END_VAR
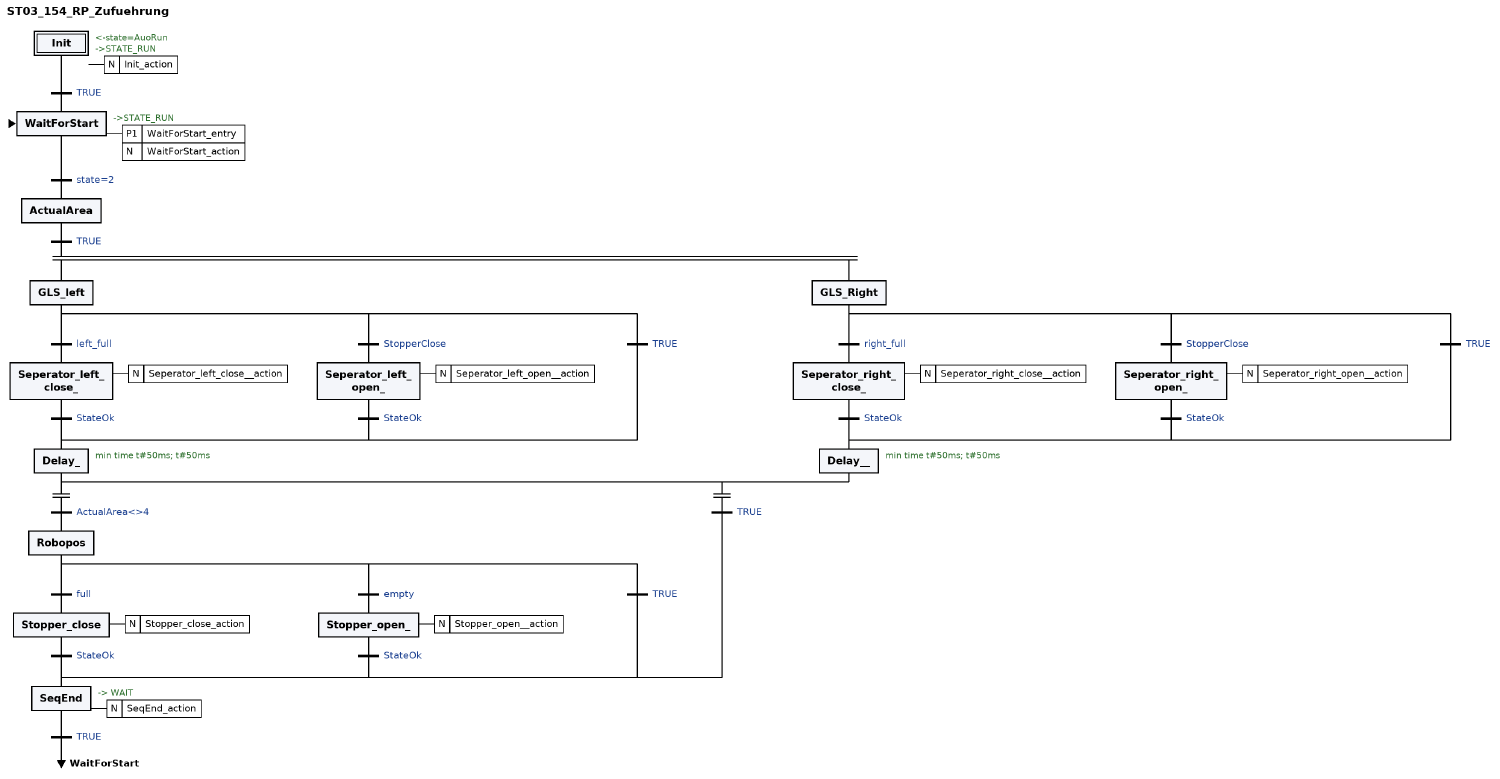
[picture p57: ST03_154_RP_Zufuehrung (SFC)]
INITIAL_STEP Init: (* <-state=AuoRun / ->STATE_RUN *)
	Init_action(N);
END_STEP
TRANSITION FROM Init TO WaitForStart := TRUE;
END_TRANSITION
STEP WaitForStart: (* ->STATE_RUN *)
	WaitForStart_entry(P1);
	WaitForStart_action(N);
END_STEP
TRANSITION FROM WaitForStart TO ActualArea := state=2;
END_TRANSITION
STEP ActualArea:
END_STEP
TRANSITION FROM ActualArea TO (GLS_left, GLS_Right) := TRUE;
END_TRANSITION
STEP GLS_left:
END_STEP
TRANSITION FROM GLS_left TO Seperator_left_close_ := left_full;
END_TRANSITION
TRANSITION FROM GLS_left TO Seperator_left_open_ := StopperClose;
END_TRANSITION
TRANSITION FROM GLS_left TO Delay_ := TRUE;
END_TRANSITION
STEP Seperator_left_close_:
	Seperator_left_close__action(N);
END_STEP
TRANSITION FROM Seperator_left_close_ TO Delay_ := StateOk;
END_TRANSITION
STEP Seperator_left_open_:
	Seperator_left_open__action(N);
END_STEP
TRANSITION FROM Seperator_left_open_ TO Delay_ := StateOk;
END_TRANSITION
STEP Delay_: (* min time t#50ms; t#50ms *)
END_STEP
STEP GLS_Right:
END_STEP
TRANSITION FROM GLS_Right TO Seperator_right_close_ := right_full;
END_TRANSITION
TRANSITION FROM GLS_Right TO Seperator_right_open_ := StopperClose;
END_TRANSITION
TRANSITION FROM GLS_Right TO Delay__ := TRUE;
END_TRANSITION
STEP Seperator_right_close_:
	Seperator_right_close__action(N);
END_STEP
TRANSITION FROM Seperator_right_close_ TO Delay__ := StateOk;
END_TRANSITION
STEP Seperator_right_open_:
	Seperator_right_open__action(N);
END_STEP
TRANSITION FROM Seperator_right_open_ TO Delay__ := StateOk;
END_TRANSITION
STEP Delay__: (* min time t#50ms; t#50ms *)
END_STEP
TRANSITION FROM (Delay_, Delay__) TO Robopos := ActualArea<>4;
END_TRANSITION
TRANSITION FROM (Delay_, Delay__) TO SeqEnd := TRUE;
END_TRANSITION
STEP Robopos:
END_STEP
TRANSITION FROM Robopos TO Stopper_close := full;
END_TRANSITION
TRANSITION FROM Robopos TO Stopper_open_ := empty;
END_TRANSITION
TRANSITION FROM Robopos TO SeqEnd := TRUE;
END_TRANSITION
STEP Stopper_close:
	Stopper_close_action(N);
END_STEP
TRANSITION FROM Stopper_close TO SeqEnd := StateOk;
END_TRANSITION
STEP Stopper_open_:
	Stopper_open__action(N);
END_STEP
TRANSITION FROM Stopper_open_ TO SeqEnd := StateOk;
END_TRANSITION
STEP SeqEnd: (* -> WAIT *)
	SeqEnd_action(N);
END_STEP
TRANSITION FROM SeqEnd TO WaitForStart := TRUE;
END_TRANSITION

ACTION Init_action:
Start:=FALSE;
State:=STATE_WAIT;
MsgOK:=FALSE;
MsgCancel:=FALSE;
SFCRun:=FALSE;
Result:=RESULT_NON;
END_ACTION

ACTION WaitForStart_entry:
;
END_ACTION

ACTION WaitForStart_action:
IF 	Start   THEN
	State:=STATE_RUN;
	Result:=RESULT_NON;
	SFCTimeStart:=TIME();
	Start:=FALSE;
ELSE
	State:=STATE_WAIT;
	MsgOK:=FALSE;
	MsgCancel:=FALSE;
	SFCRun:=FALSE;
END_IF
END_ACTION

ACTION Seperator_left_close__action:
ST03_419_Y61_5.MoveWork:=TRUE;	(* Förderband linke Zuführung Vereinzler AST/GST *)
END_ACTION

ACTION Seperator_left_open__action:
ST03_419_Y61_5.MoveInit:=TRUE;		(* Förderband linke Zuführung Vereinzler AST/GST *)
END_ACTION

ACTION Seperator_right_close__action:
ST03_419_Y61_6.MoveWork:=TRUE;	(* Förderband rechts Zuführung Vereinzler AST/GST *)
END_ACTION

ACTION Seperator_right_open__action:
ST03_419_Y61_6.MoveInit:=TRUE;			(* Förderband rechts Zuführung Vereinzler AST/GST *)
END_ACTION

ACTION Stopper_close_action:
ST03_419_Y61_7.MoveInit:=TRUE;		(* Förderband links/rechts Züführung Stopper AST/GST *)
END_ACTION

ACTION Stopper_open__action:
ST03_419_Y61_7.MoveWork:=TRUE;		(* Förderband links/rechts Züführung Stopper AST/GST *)
END_ACTION

ACTION SeqEnd_action:
SFCTime:=TIME_TO_DINT(TIME()-SFCTimeStart);
State:=STATE_WAIT;
END_ACTION

TRANSITION left_full:
ST03_419_B61_0.BitInToCheck			(*  Förderband Zuführung links ISK anwesend zum Vereinzeln*)
END_TRANSITION

TRANSITION StateOk:
ST03_419_Y61_5.State=STATE_OK
AND
gTipImp
END_TRANSITION

TRANSITION StopperClose:
NOT ST03_418_B60_4.ValveSensor AND
ST03_418_B60_5.ValveSensor
END_TRANSITION

TRANSITION StateOk:
ST03_419_Y61_5.State=STATE_OK 	(* Förderband  Zuführung Vereinzler AST/GST *)
AND
gTipImp
END_TRANSITION

TRANSITION right_full:
ST03_419_B61_1.BitInToCheck			(*  Förderband Zuführung rechts ISK anwesend zum Vereinzeln*)
END_TRANSITION

TRANSITION StateOk:
ST03_419_Y61_6.State=STATE_OK (* Förderband rechts Zuführung Vereinzler AST/GST *)
AND
gTipImp
END_TRANSITION

TRANSITION StopperClose:
NOT ST03_418_B60_4.ValveSensor AND
ST03_418_B60_5.ValveSensor
END_TRANSITION

TRANSITION StateOk:
ST03_419_Y61_6.State=STATE_OK 	(* Förderband rechts Zuführung Vereinzler AST/GST *)
AND
gTipImp
END_TRANSITION

TRANSITION ActualArea<>4:
Robot01.ActualArea <> 4
END_TRANSITION

TRANSITION full:
ST03_419_B61_2.BitInToCheck AND 	(*  Züführung links ISK auf Übergabeposition Roboter Palettierer*)
ST03_419_B61_3.BitInToCheck		(*  Züführung rechts ISK auf Übergabeposition Roboter Palettierer*)
END_TRANSITION

TRANSITION StateOk:
ST03_419_Y61_7.State=STATE_OK 	(* Förderband  Zuführung Vereinzler AST/GST *)
AND
gTipImp
END_TRANSITION

TRANSITION empty:
NOT ST03_419_B61_2.BitInToCheck AND 	(*  Züführung links ISK auf Übergabeposition Roboter Palettierer*)
NOT ST03_419_B61_3.BitInToCheck		(*  Züführung rechts ISK auf Übergabeposition Roboter Palettierer*)
END_TRANSITION

TRANSITION StateOk:
ST03_419_Y61_7.State=STATE_OK 	(* Förderband  Zuführung Vereinzler AST/GST *)
AND
gTipImp
END_TRANSITION
END_PROGRAM

(* POU Stations/ST_03_Ruestsaetze/ST_03_SFCs/Zufuehrungen/ST03_206pol_Zufuehrung, SFC *)
 PROGRAM ST03_206pol_Zufuehrung
VAR_OUTPUT
	SFCCurrentPOU			: STRING:='ST03_206pol_Zufuehrung';
	SFCCurrentStep			: STRING:='';
	FB_CurrentStepHistorie	: FB_CurrentStepHistorie;
	SFCTime					: DINT;
	State   				: StateObject	:= STATE_WAIT;
	Result  				: StateResult;
END_VAR
VAR_INPUT
	Start					:BOOL;
END_VAR
VAR
	MsgOK				: BOOL;
	MsgCancel			: BOOL;
	SFCRun				: BOOL;
	SFCTimeStart		: TIME;
	Delay				: TON;
	(* Userdefinded area *)

END_VAR
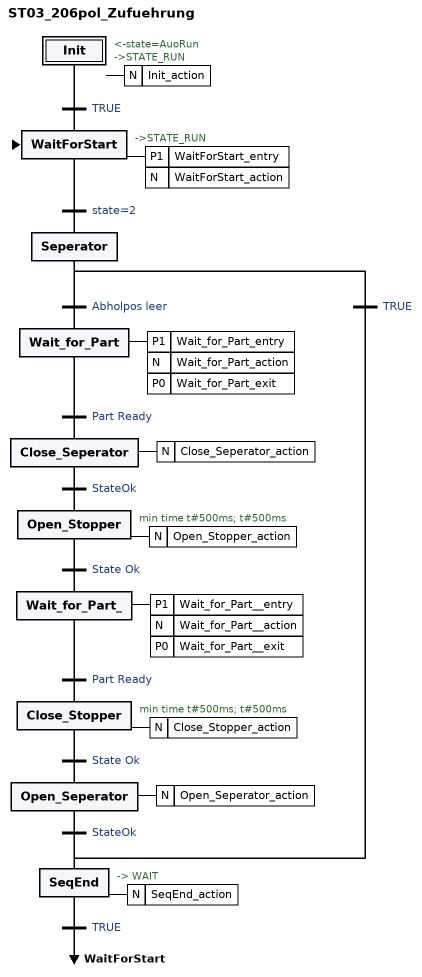
INITIAL_STEP Init: (* <-state=AuoRun / ->STATE_RUN *)
	Init_action(N);
END_STEP
TRANSITION FROM Init TO WaitForStart := TRUE;
END_TRANSITION
STEP WaitForStart: (* ->STATE_RUN *)
	WaitForStart_entry(P1);
	WaitForStart_action(N);
END_STEP
TRANSITION FROM WaitForStart TO Seperator := state=2;
END_TRANSITION
STEP Seperator:
END_STEP
TRANSITION FROM Seperator TO Wait_for_Part := Abholpos leer;
END_TRANSITION
TRANSITION FROM Seperator TO SeqEnd := TRUE;
END_TRANSITION
STEP Wait_for_Part:
	Wait_for_Part_entry(P1);
	Wait_for_Part_action(N);
	Wait_for_Part_exit(P0);
END_STEP
TRANSITION FROM Wait_for_Part TO Close_Seperator := Part Ready;
END_TRANSITION
STEP Close_Seperator:
	Close_Seperator_action(N);
END_STEP
TRANSITION FROM Close_Seperator TO Open_Stopper := StateOk;
END_TRANSITION
STEP Open_Stopper: (* min time t#500ms; t#500ms *)
	Open_Stopper_action(N);
END_STEP
TRANSITION FROM Open_Stopper TO Wait_for_Part_ := State Ok;
END_TRANSITION
STEP Wait_for_Part_:
	Wait_for_Part__entry(P1);
	Wait_for_Part__action(N);
	Wait_for_Part__exit(P0);
END_STEP
TRANSITION FROM Wait_for_Part_ TO Close_Stopper := Part Ready;
END_TRANSITION
STEP Close_Stopper: (* min time t#500ms; t#500ms *)
	Close_Stopper_action(N);
END_STEP
TRANSITION FROM Close_Stopper TO Open_Seperator := State Ok;
END_TRANSITION
STEP Open_Seperator:
	Open_Seperator_action(N);
END_STEP
TRANSITION FROM Open_Seperator TO SeqEnd := StateOk;
END_TRANSITION
STEP SeqEnd: (* -> WAIT *)
	SeqEnd_action(N);
END_STEP
TRANSITION FROM SeqEnd TO WaitForStart := TRUE;
END_TRANSITION

ACTION Init_action:
Start:=FALSE;
State:=STATE_WAIT;
MsgOK:=FALSE;
MsgCancel:=FALSE;
SFCRun:=FALSE;
Result:=RESULT_NON;
END_ACTION

ACTION WaitForStart_entry:
;
END_ACTION

ACTION WaitForStart_action:
IF 	Start   THEN
	State:=STATE_RUN;
	Result:=RESULT_NON;
	SFCTimeStart:=TIME();
	Start:=FALSE;
ELSE
	State:=STATE_WAIT;
	MsgOK:=FALSE;
	MsgCancel:=FALSE;
	SFCRun:=FALSE;
END_IF
END_ACTION

ACTION Wait_for_Part_entry:
ProcessMessage01:='';
Delay.IN:=FALSE;
Delay();
END_ACTION

ACTION Wait_for_Part_action:
ProcessMessage01:='1IM6';(*warte auf Teil in Vereinzelung*)
Delay.IN:=ST03_435_B67_7.BitInToCheck; 		 (* Schnittstelle Iso auf Übergabeposition *)
Delay.PT:=T#500ms;
Delay();
END_ACTION

ACTION Wait_for_Part_exit:
ProcessMessage01:='';
END_ACTION

ACTION Close_Seperator_action:
ST03_437_Y68_5.MoveWork:=TRUE;		(* Förderband  Zuführung Vereinzler AST/GST *)
END_ACTION

ACTION Open_Stopper_action:
ST03_437_Y68_6.MoveWork:=TRUE;		(* Förderband  Züführung Stopper AST/GST *)
END_ACTION

ACTION Wait_for_Part__entry:
ProcessMessage01:='';
Delay.IN:=FALSE;
Delay();
END_ACTION

ACTION Wait_for_Part__action:
ProcessMessage01:='1IM6';(*warte auf Teil in Vereinzelung*)
Delay.IN:=	ST03_Init_AbholPos.RoboPos31 OR
			ST03_Init_AbholPos.RoboPos35 OR
			NOT ST03_437_B68_4.BitInToCheck;
Delay.PT:=T#500ms;
Delay();
END_ACTION

ACTION Wait_for_Part__exit:
ProcessMessage01:='';
END_ACTION

ACTION Close_Stopper_action:
ST03_437_Y68_6.MoveInit:=TRUE;		(* Förderband  Züführung Stopper AST/GST *)
END_ACTION

ACTION Open_Seperator_action:
ST03_437_Y68_5.MoveInit:=TRUE;		(* Förderband  Zuführung Vereinzler AST/GST *)
END_ACTION

ACTION SeqEnd_action:
SFCTime:=TIME_TO_DINT(TIME()-SFCTimeStart);
State:=STATE_WAIT;
END_ACTION

TRANSITION Abholpos leer:
NOT ST03_Init_AbholPos.RoboPos31 AND
NOT ST03_Init_AbholPos.RoboPos35
END_TRANSITION

TRANSITION Part Ready:
Delay.Q AND
ST03_435_B67_7.BitInToCheck	AND	(*  ISK anwesend am Stoper*)
Robot01.ActualArea <> 4
END_TRANSITION

TRANSITION StateOk:
ST03_437_Y68_5.State=STATE_OK 	(* Förderband  Zuführung Vereinzler AST/GST *)

(*ST03_426_B68_4.BitInToCheck	AND		(*  Züführung  ISK auf Übergabeposition Roboter Palettierer*)
NOT ST03_425_B67_7.BitInToCheck AND	(*  ISK anwesend am Vereinzler*)
gTipImp*)
END_TRANSITION

TRANSITION State Ok:
ST03_437_Y68_6.State=STATE_OK 	(* Förderband  Züführung Stopper AST/GST *)
END_TRANSITION

TRANSITION Part Ready:
Delay.Q AND
(ST03_Init_AbholPos.RoboPos31 OR
ST03_Init_AbholPos.RoboPos35) AND
Robot01.ActualArea <> 4
END_TRANSITION

TRANSITION State Ok:
ST03_437_Y68_6.State=STATE_OK 	(* Förderband  Züführung Stopper AST/GST *)
END_TRANSITION

TRANSITION StateOk:
ST03_437_Y68_5.State=STATE_OK 	(* Förderband  Zuführung Vereinzler AST/GST *)
END_TRANSITION
END_PROGRAM

(* POU Stations/ST_03_Ruestsaetze/ST_03_SFCs/Zufuehrungen/ST03_92pol_Zufuehrung, SFC *)
 PROGRAM ST03_92pol_Zufuehrung
VAR_OUTPUT
	SFCCurrentPOU			: STRING:='ST03_92pol_Zufuehrung';
	SFCCurrentStep			: STRING:='';
	FB_CurrentStepHistorie	: FB_CurrentStepHistorie;
	SFCTime					: DINT;
	State   				: StateObject	:= STATE_WAIT;
	Result  				: StateResult;
END_VAR
VAR_INPUT
	Start					:BOOL;
END_VAR
VAR
	MsgOK				: BOOL;
	MsgCancel			: BOOL;
	SFCRun				: BOOL;
	SFCTimeStart		: TIME;
	Delay				: TON;
	(* Userdefinded area *)

END_VAR
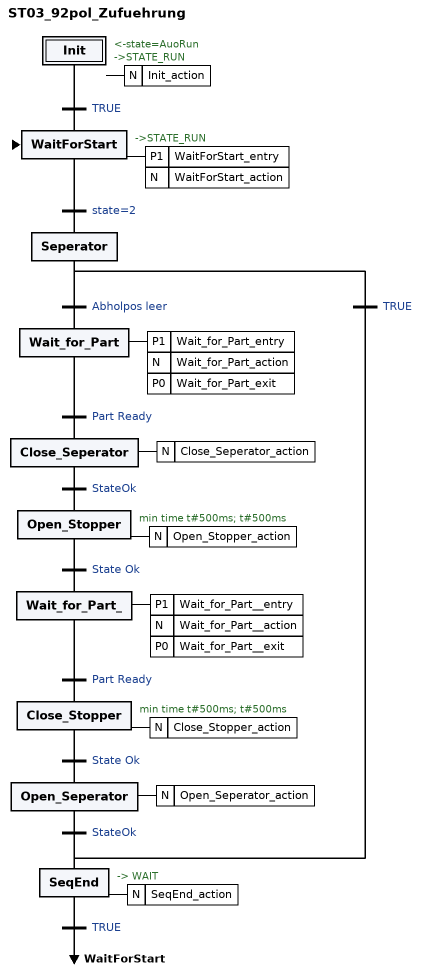
INITIAL_STEP Init: (* <-state=AuoRun / ->STATE_RUN *)
	Init_action(N);
END_STEP
TRANSITION FROM Init TO WaitForStart := TRUE;
END_TRANSITION
STEP WaitForStart: (* ->STATE_RUN *)
	WaitForStart_entry(P1);
	WaitForStart_action(N);
END_STEP
TRANSITION FROM WaitForStart TO Seperator := state=2;
END_TRANSITION
STEP Seperator:
END_STEP
TRANSITION FROM Seperator TO Wait_for_Part := Abholpos leer;
END_TRANSITION
TRANSITION FROM Seperator TO SeqEnd := TRUE;
END_TRANSITION
STEP Wait_for_Part:
	Wait_for_Part_entry(P1);
	Wait_for_Part_action(N);
	Wait_for_Part_exit(P0);
END_STEP
TRANSITION FROM Wait_for_Part TO Close_Seperator := Part Ready;
END_TRANSITION
STEP Close_Seperator:
	Close_Seperator_action(N);
END_STEP
TRANSITION FROM Close_Seperator TO Open_Stopper := StateOk;
END_TRANSITION
STEP Open_Stopper: (* min time t#500ms; t#500ms *)
	Open_Stopper_action(N);
END_STEP
TRANSITION FROM Open_Stopper TO Wait_for_Part_ := State Ok;
END_TRANSITION
STEP Wait_for_Part_:
	Wait_for_Part__entry(P1);
	Wait_for_Part__action(N);
	Wait_for_Part__exit(P0);
END_STEP
TRANSITION FROM Wait_for_Part_ TO Close_Stopper := Part Ready;
END_TRANSITION
STEP Close_Stopper: (* min time t#500ms; t#500ms *)
	Close_Stopper_action(N);
END_STEP
TRANSITION FROM Close_Stopper TO Open_Seperator := State Ok;
END_TRANSITION
STEP Open_Seperator:
	Open_Seperator_action(N);
END_STEP
TRANSITION FROM Open_Seperator TO SeqEnd := StateOk;
END_TRANSITION
STEP SeqEnd: (* -> WAIT *)
	SeqEnd_action(N);
END_STEP
TRANSITION FROM SeqEnd TO WaitForStart := TRUE;
END_TRANSITION

ACTION Init_action:
Start:=FALSE;
State:=STATE_WAIT;
MsgOK:=FALSE;
MsgCancel:=FALSE;
SFCRun:=FALSE;
Result:=RESULT_NON;
END_ACTION

ACTION WaitForStart_entry:
;
END_ACTION

ACTION WaitForStart_action:
IF 	Start   THEN
	State:=STATE_RUN;
	Result:=RESULT_NON;
	SFCTimeStart:=TIME();
	Start:=FALSE;
ELSE
	State:=STATE_WAIT;
	MsgOK:=FALSE;
	MsgCancel:=FALSE;
	SFCRun:=FALSE;
END_IF
END_ACTION

ACTION Wait_for_Part_entry:
ProcessMessage01:='';
Delay.IN:=FALSE;
Delay();
END_ACTION

ACTION Wait_for_Part_action:
ProcessMessage01:='1IM6';(*warte auf Teil in Vereinzelung*)
Delay.IN:=ST03_444_B69_7.BitInToCheck; 		 (* Schnittstelle Iso auf Übergabeposition *)
Delay.PT:=T#500ms;
Delay();
END_ACTION

ACTION Wait_for_Part_exit:
ProcessMessage01:='';
END_ACTION

ACTION Close_Seperator_action:
ST03_446_Y70_5.MoveWork:=TRUE;		(* Förderband  Zuführung Vereinzler AST/GST *)
END_ACTION

ACTION Open_Stopper_action:
ST03_446_Y70_6.MoveWork:=TRUE;		(* Förderband  Züführung Stopper AST/GST *)
END_ACTION

ACTION Wait_for_Part__entry:
ProcessMessage01:='';
Delay.IN:=FALSE;
Delay();
END_ACTION

ACTION Wait_for_Part__action:
ProcessMessage01:='1IM6';(*warte auf Teil in Vereinzelung*)
Delay.IN:=ST03_446_B70_4.BitInToCheck; 		 (* Schnittstelle Iso auf Übergabeposition Roboter *)
Delay.PT:=T#500ms;
Delay();
END_ACTION

ACTION Wait_for_Part__exit:
ProcessMessage01:='';
END_ACTION

ACTION Close_Stopper_action:
ST03_446_Y70_6.MoveInit:=TRUE;		(* Förderband  Züführung Stopper AST/GST *)
END_ACTION

ACTION Open_Seperator_action:
ST03_446_Y70_5.MoveInit:=TRUE;		(* Förderband  Zuführung Vereinzler AST/GST *)
END_ACTION

ACTION SeqEnd_action:
SFCTime:=TIME_TO_DINT(TIME()-SFCTimeStart);
State:=STATE_WAIT;
END_ACTION

TRANSITION Abholpos leer:
NOT  ST03_446_B70_4.BitInToCheck
END_TRANSITION

TRANSITION Part Ready:
Delay.Q AND
NOT ST03_446_B70_4.BitInToCheck	AND		(*  Züführung  ISK auf Übergabeposition Roboter Palettierer*)
ST03_444_B69_7.BitInToCheck	AND	(*  ISK anwesend am Vereinzler*)
Robot01.ActualArea <> 4
END_TRANSITION

TRANSITION StateOk:
ST03_446_Y70_5.State=STATE_OK 	(* Förderband  Zuführung Vereinzler AST/GST *)

(*ST03_426_B68_4.BitInToCheck	AND		(*  Züführung  ISK auf Übergabeposition Roboter Palettierer*)
NOT ST03_425_B67_7.BitInToCheck AND	(*  ISK anwesend am Vereinzler*)
gTipImp*)
END_TRANSITION

TRANSITION State Ok:
ST03_446_Y70_6.State=STATE_OK 	(* Förderband  Züführung Stopper AST/GST *)
END_TRANSITION

TRANSITION Part Ready:
Delay.Q AND
(*NOT ST03_426_B68_4.BitInToCheck	AND		(*  Züführung  ISK auf Übergabeposition Roboter Palettierer*)
ST03_425_B67_7.BitInToCheck	AND*)	(*  ISK anwesend am Vereinzler*)
Robot01.ActualArea <> 4
END_TRANSITION

TRANSITION State Ok:
ST03_446_Y70_6.State=STATE_OK 	(* Förderband  Züführung Stopper AST/GST *)
END_TRANSITION

TRANSITION StateOk:
ST03_446_Y70_5.State=STATE_OK 	(* Förderband  Zuführung Vereinzler AST/GST *)

(*ST03_426_B68_4.BitInToCheck	AND		(*  Züführung  ISK auf Übergabeposition Roboter Palettierer*)
NOT ST03_425_B67_7.BitInToCheck AND	(*  ISK anwesend am Vereinzler*)
gTipImp*)
END_TRANSITION
END_PROGRAM

(* POU Stations/ST_03_Ruestsaetze/ST_03_SFCs/Zufuehrungen/ST03_124pol_Zufuehrung, SFC *)
 PROGRAM ST03_124pol_Zufuehrung
VAR_OUTPUT
	SFCCurrentPOU			: STRING:='ST03_124pol_Zufuehrung';
	SFCCurrentStep			: STRING:='';
	FB_CurrentStepHistorie	: FB_CurrentStepHistorie;
	SFCTime					: DINT;
	State   				: StateObject	:= STATE_WAIT;
	Result  				: StateResult;
END_VAR
VAR_INPUT
	Start					:BOOL;
END_VAR
VAR
	MsgOK				: BOOL;
	MsgCancel			: BOOL;
	SFCRun				: BOOL;
	SFCTimeStart		: TIME;
	Delay				: TON;
	(* Userdefinded area *)

END_VAR
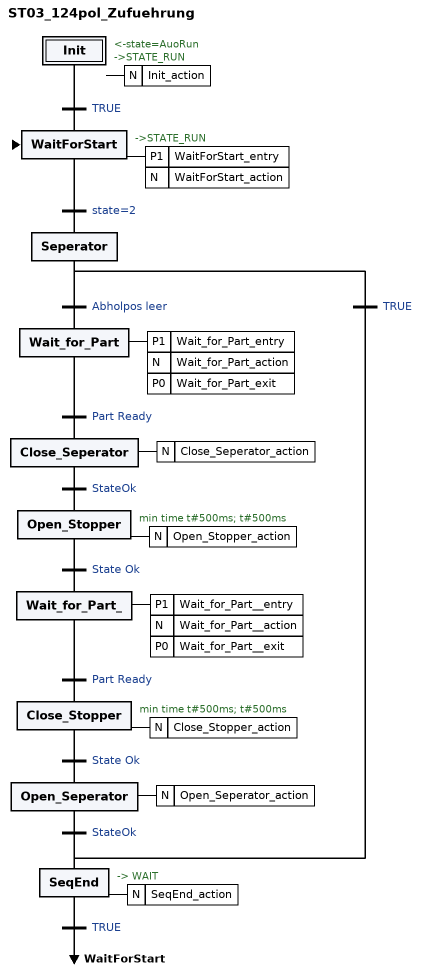
INITIAL_STEP Init: (* <-state=AuoRun / ->STATE_RUN *)
	Init_action(N);
END_STEP
TRANSITION FROM Init TO WaitForStart := TRUE;
END_TRANSITION
STEP WaitForStart: (* ->STATE_RUN *)
	WaitForStart_entry(P1);
	WaitForStart_action(N);
END_STEP
TRANSITION FROM WaitForStart TO Seperator := state=2;
END_TRANSITION
STEP Seperator:
END_STEP
TRANSITION FROM Seperator TO Wait_for_Part := Abholpos leer;
END_TRANSITION
TRANSITION FROM Seperator TO SeqEnd := TRUE;
END_TRANSITION
STEP Wait_for_Part:
	Wait_for_Part_entry(P1);
	Wait_for_Part_action(N);
	Wait_for_Part_exit(P0);
END_STEP
TRANSITION FROM Wait_for_Part TO Close_Seperator := Part Ready;
END_TRANSITION
STEP Close_Seperator:
	Close_Seperator_action(N);
END_STEP
TRANSITION FROM Close_Seperator TO Open_Stopper := StateOk;
END_TRANSITION
STEP Open_Stopper: (* min time t#500ms; t#500ms *)
	Open_Stopper_action(N);
END_STEP
TRANSITION FROM Open_Stopper TO Wait_for_Part_ := State Ok;
END_TRANSITION
STEP Wait_for_Part_:
	Wait_for_Part__entry(P1);
	Wait_for_Part__action(N);
	Wait_for_Part__exit(P0);
END_STEP
TRANSITION FROM Wait_for_Part_ TO Close_Stopper := Part Ready;
END_TRANSITION
STEP Close_Stopper: (* min time t#500ms; t#500ms *)
	Close_Stopper_action(N);
END_STEP
TRANSITION FROM Close_Stopper TO Open_Seperator := State Ok;
END_TRANSITION
STEP Open_Seperator:
	Open_Seperator_action(N);
END_STEP
TRANSITION FROM Open_Seperator TO SeqEnd := StateOk;
END_TRANSITION
STEP SeqEnd: (* -> WAIT *)
	SeqEnd_action(N);
END_STEP
TRANSITION FROM SeqEnd TO WaitForStart := TRUE;
END_TRANSITION

ACTION Init_action:
Start:=FALSE;
State:=STATE_WAIT;
MsgOK:=FALSE;
MsgCancel:=FALSE;
SFCRun:=FALSE;
Result:=RESULT_NON;
END_ACTION

ACTION WaitForStart_entry:
;
END_ACTION

ACTION WaitForStart_action:
IF 	Start   THEN
	State:=STATE_RUN;
	Result:=RESULT_NON;
	SFCTimeStart:=TIME();
	Start:=FALSE;
ELSE
	State:=STATE_WAIT;
	MsgOK:=FALSE;
	MsgCancel:=FALSE;
	SFCRun:=FALSE;
END_IF
END_ACTION

ACTION Wait_for_Part_entry:
ProcessMessage01:='';
Delay.IN:=FALSE;
Delay();
END_ACTION

ACTION Wait_for_Part_action:
ProcessMessage01:='1IM6';(*warte auf Teil in Vereinzelung*)
Delay.IN:=ST03_451_B69_7.BitInToCheck; 		 (* Schnittstelle Iso auf Übergabeposition *)
Delay.PT:=T#500ms;
Delay();
END_ACTION

ACTION Wait_for_Part_exit:
ProcessMessage01:='';
END_ACTION

ACTION Close_Seperator_action:
ST03_453_Y70_5.MoveWork:=TRUE;		(* Förderband  Zuführung Vereinzler AST/GST *)
END_ACTION

ACTION Open_Stopper_action:
ST03_453_Y70_6.MoveWork:=TRUE;		(* Förderband  Züführung Stopper AST/GST *)
END_ACTION

ACTION Wait_for_Part__entry:
ProcessMessage01:='';
Delay.IN:=FALSE;
Delay();
END_ACTION

ACTION Wait_for_Part__action:
ProcessMessage01:='1IM6';(*warte auf Teil in Vereinzelung*)
Delay.IN:=ST03_453_B70_4.BitInToCheck; 		 (* Schnittstelle Iso auf Übergabeposition Roboter *)
Delay.PT:=T#500ms;
Delay();
END_ACTION

ACTION Wait_for_Part__exit:
ProcessMessage01:='';
END_ACTION

ACTION Close_Stopper_action:
ST03_453_Y70_6.MoveInit:=TRUE;		(* Förderband  Züführung Stopper AST/GST *)
END_ACTION

ACTION Open_Seperator_action:
ST03_453_Y70_5.MoveInit:=TRUE;		(* Förderband  Zuführung Vereinzler AST/GST *)
END_ACTION

ACTION SeqEnd_action:
SFCTime:=TIME_TO_DINT(TIME()-SFCTimeStart);
State:=STATE_WAIT;
END_ACTION

TRANSITION Abholpos leer:
NOT  ST03_453_B70_4.BitInToCheck
END_TRANSITION

TRANSITION Part Ready:
Delay.Q AND
NOT ST03_453_B70_4.BitInToCheck	AND		(*  Züführung  ISK auf Übergabeposition Roboter Palettierer*)
ST03_451_B69_7.BitInToCheck	AND	(*  ISK anwesend am Vereinzler*)
Robot01.ActualArea <> 4
END_TRANSITION

TRANSITION StateOk:
ST03_453_Y70_5.State=STATE_OK 	(* Förderband  Zuführung Vereinzler AST/GST *)

(*ST03_426_B68_4.BitInToCheck	AND		(*  Züführung  ISK auf Übergabeposition Roboter Palettierer*)
NOT ST03_425_B67_7.BitInToCheck AND	(*  ISK anwesend am Vereinzler*)
gTipImp*)
END_TRANSITION

TRANSITION State Ok:
ST03_453_Y70_6.State=STATE_OK 	(* Förderband  Züführung Stopper AST/GST *)
END_TRANSITION

TRANSITION Part Ready:
Delay.Q AND
(*NOT ST03_426_B68_4.BitInToCheck	AND		(*  Züführung  ISK auf Übergabeposition Roboter Palettierer*)
ST03_425_B67_7.BitInToCheck	AND*)	(*  ISK anwesend am Vereinzler*)
Robot01.ActualArea <> 4
END_TRANSITION

TRANSITION State Ok:
ST03_453_Y70_6.State=STATE_OK 	(* Förderband  Züführung Stopper AST/GST *)
END_TRANSITION

TRANSITION StateOk:
ST03_453_Y70_5.State=STATE_OK 	(* Förderband  Zuführung Vereinzler AST/GST *)

(*ST03_426_B68_4.BitInToCheck	AND		(*  Züführung  ISK auf Übergabeposition Roboter Palettierer*)
NOT ST03_425_B67_7.BitInToCheck AND	(*  ISK anwesend am Vereinzler*)
gTipImp*)
END_TRANSITION
END_PROGRAM

(* POU Stations/ST_03_Ruestsaetze/ST_03_SFCs/Zufuehrungen/ST03_46pol_Zufuehrung, SFC *)
 PROGRAM ST03_46pol_Zufuehrung
VAR_OUTPUT
	SFCCurrentPOU			: STRING:='ST03_46pol_Zufuehrung';
	SFCCurrentStep			: STRING:='';
	FB_CurrentStepHistorie	: FB_CurrentStepHistorie;
	SFCTime					: DINT;
	State   				: StateObject	:= STATE_WAIT;
	Result  				: StateResult;
END_VAR
VAR_INPUT
	Start					:BOOL;
END_VAR
VAR
	MsgOK				: BOOL;
	MsgCancel			: BOOL;
	SFCRun				: BOOL;
	SFCTimeStart		: TIME;
	Delay				: TON;
	(* Userdefinded area *)

END_VAR
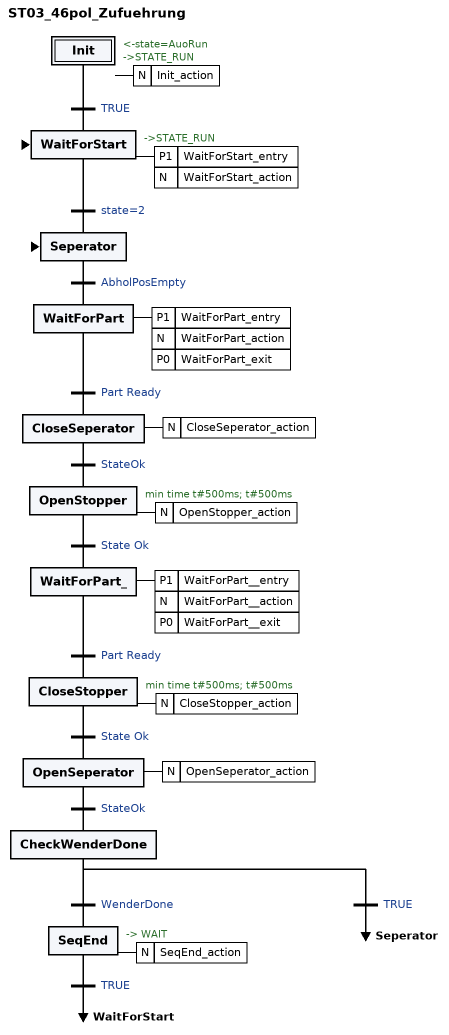
INITIAL_STEP Init: (* <-state=AuoRun / ->STATE_RUN *)
	Init_action(N);
END_STEP
TRANSITION FROM Init TO WaitForStart := TRUE;
END_TRANSITION
STEP WaitForStart: (* ->STATE_RUN *)
	WaitForStart_entry(P1);
	WaitForStart_action(N);
END_STEP
TRANSITION FROM WaitForStart TO Seperator := state=2;
END_TRANSITION
STEP Seperator:
END_STEP
TRANSITION FROM Seperator TO WaitForPart := AbholPosEmpty;
END_TRANSITION
STEP WaitForPart:
	WaitForPart_entry(P1);
	WaitForPart_action(N);
	WaitForPart_exit(P0);
END_STEP
TRANSITION FROM WaitForPart TO CloseSeperator := Part Ready;
END_TRANSITION
STEP CloseSeperator:
	CloseSeperator_action(N);
END_STEP
TRANSITION FROM CloseSeperator TO OpenStopper := StateOk;
END_TRANSITION
STEP OpenStopper: (* min time t#500ms; t#500ms *)
	OpenStopper_action(N);
END_STEP
TRANSITION FROM OpenStopper TO WaitForPart_ := State Ok;
END_TRANSITION
STEP WaitForPart_:
	WaitForPart__entry(P1);
	WaitForPart__action(N);
	WaitForPart__exit(P0);
END_STEP
TRANSITION FROM WaitForPart_ TO CloseStopper := Part Ready;
END_TRANSITION
STEP CloseStopper: (* min time t#500ms; t#500ms *)
	CloseStopper_action(N);
END_STEP
TRANSITION FROM CloseStopper TO OpenSeperator := State Ok;
END_TRANSITION
STEP OpenSeperator:
	OpenSeperator_action(N);
END_STEP
TRANSITION FROM OpenSeperator TO CheckWenderDone := StateOk;
END_TRANSITION
STEP CheckWenderDone:
END_STEP
TRANSITION FROM CheckWenderDone TO SeqEnd := WenderDone;
END_TRANSITION
TRANSITION FROM CheckWenderDone TO Seperator := TRUE;
END_TRANSITION
STEP SeqEnd: (* -> WAIT *)
	SeqEnd_action(N);
END_STEP
TRANSITION FROM SeqEnd TO WaitForStart := TRUE;
END_TRANSITION

ACTION Init_action:
Start:=FALSE;
State:=STATE_WAIT;
MsgOK:=FALSE;
MsgCancel:=FALSE;
SFCRun:=FALSE;
Result:=RESULT_NON;
END_ACTION

ACTION WaitForStart_entry:
;
END_ACTION

ACTION WaitForStart_action:
IF 	Start   THEN
	State:=STATE_RUN;
	Result:=RESULT_NON;
	SFCTimeStart:=TIME();
	Start:=FALSE;
ELSE
	State:=STATE_WAIT;
	MsgOK:=FALSE;
	MsgCancel:=FALSE;
	SFCRun:=FALSE;
END_IF
END_ACTION

ACTION WaitForPart_entry:
ProcessMessage01:='';
Delay.IN:=FALSE;
Delay();
END_ACTION

ACTION WaitForPart_action:
ProcessMessage01:='1IM6';(*warte auf Teil in Vereinzelung*)
Delay.IN:=ST03_461_B69_7.BitInToCheck; 		 (*  ISK anwesend am Stopper *)
Delay.PT:=T#500ms;
Delay();
END_ACTION

ACTION WaitForPart_exit:
ProcessMessage01:='';
END_ACTION

ACTION CloseSeperator_action:
ST03_464_Y71_3.MoveWork:=TRUE;		(* Förderband  Zuführung Vereinzler AST/GST *)
END_ACTION

ACTION OpenStopper_action:
ST03_464_Y71_4.MoveWork:=TRUE;		(* Förderband  Züführung Stopper AST/GST *)
END_ACTION

ACTION WaitForPart__entry:
ProcessMessage01:='';
Delay.IN:=FALSE;
Delay();
END_ACTION

ACTION WaitForPart__action:
ProcessMessage01:='1IM6';(*warte auf Teil in Vereinzelung*)
Delay.IN:=ST03_463_B70_7.BitInToCheck; 		 (* Züführung  ISK auf Übergabeposition Roboter Palettierer  *)
Delay.PT:=T#500ms;
Delay();
END_ACTION

ACTION WaitForPart__exit:
ProcessMessage01:='';
END_ACTION

ACTION CloseStopper_action:
ST03_464_Y71_4.MoveInit:=TRUE;		(*  Förderband  Zuführung Stopper AST/GST*)
END_ACTION

ACTION OpenSeperator_action:
ST03_464_Y71_3.MoveInit:=TRUE;		(* Förderband  Zuführung Vereinzler AST/GST *)
END_ACTION

ACTION SeqEnd_action:
SFCTime:=TIME_TO_DINT(TIME()-SFCTimeStart);
State:=STATE_WAIT;
END_ACTION

TRANSITION AbholPosEmpty:
NOT  ST03_463_B70_7.BitInToCheck
END_TRANSITION

TRANSITION Part Ready:
Delay.Q AND
NOT ST03_463_B70_7.BitInToCheck	AND		(*  Züführung  ISK auf Übergabeposition Roboter Palettierer*)
ST03_461_B69_7.BitInToCheck	AND	(*  ISK anwesend am Vereinzler*)
Robot01.ActualArea <> 4
END_TRANSITION

TRANSITION StateOk:
ST03_464_Y71_3.State=STATE_OK 	(* Förderband  Zuführung Vereinzler AST/GST *)
END_TRANSITION

TRANSITION State Ok:
ST03_464_Y71_4.State=STATE_OK 	(* Förderband  Züführung Stopper AST/GST *)
END_TRANSITION

TRANSITION Part Ready:
Delay.Q AND
Robot01.ActualArea <> 4
END_TRANSITION

TRANSITION State Ok:
ST03_464_Y71_4.State=STATE_OK 	(* Förderband  Züführung Stopper AST/GST *)
END_TRANSITION

TRANSITION StateOk:
ST03_464_Y71_3.State=STATE_OK 	(* Förderband  Zuführung Vereinzler AST/GST *)
END_TRANSITION

TRANSITION WenderDone:
NOT ST03_461_B69_7.BitInToCheck			(*  ISK anwesend am Vereinzler*)
END_TRANSITION
END_PROGRAM

(* POU Stations/ST_03_Ruestsaetze/ST_03_SFCs/Zufuehrungen/ST03_46pol_Wendeeinheit, SFC *)
 PROGRAM ST03_46pol_Wendeeinheit
VAR_OUTPUT
	SFCCurrentPOU			: STRING:='ST03_46pol_Wendeeinheit';
	SFCCurrentStep			: STRING:='';
	FB_CurrentStepHistorie	: FB_CurrentStepHistorie;
	SFCTime					: DINT;
	State   				: StateObject	:= STATE_WAIT;
	Result  				: StateResult;
END_VAR
VAR_INPUT
	Start					:BOOL;
END_VAR
VAR
	MsgOK				: BOOL;
	MsgCancel			: BOOL;
	SFCRun				: BOOL;
	SFCTimeStart		: TIME;
	Delay				: TON;
	(* Userdefinded area *)
	WenderDone			: BOOL;
END_VAR
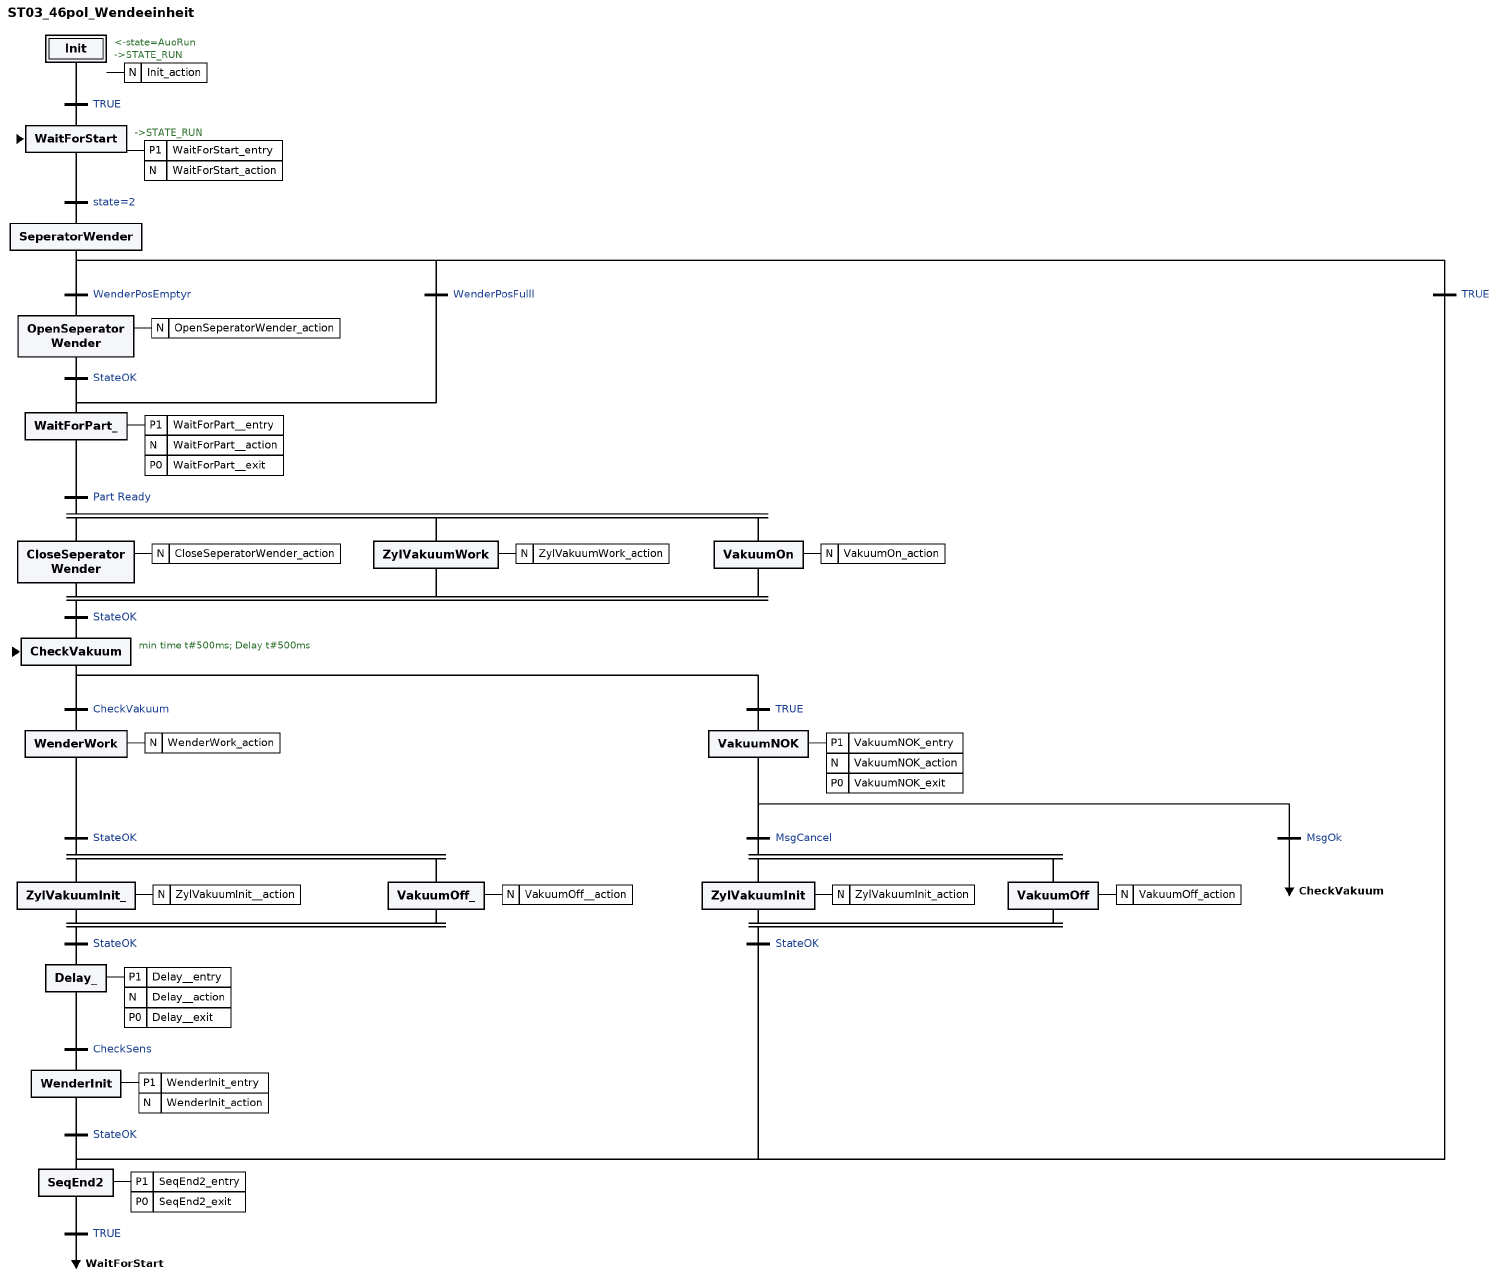
INITIAL_STEP Init: (* <-state=AuoRun / ->STATE_RUN *)
	Init_action(N);
END_STEP
TRANSITION FROM Init TO WaitForStart := TRUE;
END_TRANSITION
STEP WaitForStart: (* ->STATE_RUN *)
	WaitForStart_entry(P1);
	WaitForStart_action(N);
END_STEP
TRANSITION FROM WaitForStart TO SeperatorWender := state=2;
END_TRANSITION
STEP SeperatorWender:
END_STEP
TRANSITION FROM SeperatorWender TO OpenSeperatorWender := WenderPosEmptyr;
END_TRANSITION
TRANSITION FROM SeperatorWender TO WaitForPart_ := WenderPosFulll;
END_TRANSITION
TRANSITION FROM SeperatorWender TO SeqEnd2 := TRUE;
END_TRANSITION
STEP OpenSeperatorWender:
	OpenSeperatorWender_action(N);
END_STEP
TRANSITION FROM OpenSeperatorWender TO WaitForPart_ := StateOK;
END_TRANSITION
STEP WaitForPart_:
	WaitForPart__entry(P1);
	WaitForPart__action(N);
	WaitForPart__exit(P0);
END_STEP
TRANSITION FROM WaitForPart_ TO (CloseSeperatorWender, ZylVakuumWork, VakuumOn) := Part Ready;
END_TRANSITION
STEP CloseSeperatorWender:
	CloseSeperatorWender_action(N);
END_STEP
STEP ZylVakuumWork:
	ZylVakuumWork_action(N);
END_STEP
STEP VakuumOn:
	VakuumOn_action(N);
END_STEP
TRANSITION FROM (CloseSeperatorWender, ZylVakuumWork, VakuumOn) TO CheckVakuum := StateOK;
END_TRANSITION
STEP CheckVakuum: (* min time t#500ms; Delay t#500ms *)
END_STEP
TRANSITION FROM CheckVakuum TO WenderWork := CheckVakuum;
END_TRANSITION
TRANSITION FROM CheckVakuum TO VakuumNOK := TRUE;
END_TRANSITION
STEP WenderWork:
	WenderWork_action(N);
END_STEP
TRANSITION FROM WenderWork TO (ZylVakuumInit_, VakuumOff_) := StateOK;
END_TRANSITION
STEP ZylVakuumInit_:
	ZylVakuumInit__action(N);
END_STEP
STEP VakuumOff_:
	VakuumOff__action(N);
END_STEP
TRANSITION FROM (ZylVakuumInit_, VakuumOff_) TO Delay_ := StateOK;
END_TRANSITION
STEP Delay_:
	Delay__entry(P1);
	Delay__action(N);
	Delay__exit(P0);
END_STEP
TRANSITION FROM Delay_ TO WenderInit := CheckSens;
END_TRANSITION
STEP WenderInit:
	WenderInit_entry(P1);
	WenderInit_action(N);
END_STEP
TRANSITION FROM WenderInit TO SeqEnd2 := StateOK;
END_TRANSITION
STEP VakuumNOK:
	VakuumNOK_entry(P1);
	VakuumNOK_action(N);
	VakuumNOK_exit(P0);
END_STEP
TRANSITION FROM VakuumNOK TO (ZylVakuumInit, VakuumOff) := MsgCancel;
END_TRANSITION
TRANSITION FROM VakuumNOK TO CheckVakuum := MsgOk;
END_TRANSITION
STEP ZylVakuumInit:
	ZylVakuumInit_action(N);
END_STEP
STEP VakuumOff:
	VakuumOff_action(N);
END_STEP
TRANSITION FROM (ZylVakuumInit, VakuumOff) TO SeqEnd2 := StateOK;
END_TRANSITION
STEP SeqEnd2:
	SeqEnd2_entry(P1);
	SeqEnd2_exit(P0);
END_STEP
TRANSITION FROM SeqEnd2 TO WaitForStart := TRUE;
END_TRANSITION

ACTION Init_action:
Start:=FALSE;
State:=STATE_WAIT;
MsgOK:=FALSE;
MsgCancel:=FALSE;
SFCRun:=FALSE;
Result:=RESULT_NON;
END_ACTION

ACTION WaitForStart_entry:
;
END_ACTION

ACTION WaitForStart_action:
IF 	Start   THEN
	State:=STATE_RUN;
	Result:=RESULT_NON;
	SFCTimeStart:=TIME();
	Start:=FALSE;
	WenderDone:=FALSE;
ELSE
	State:=STATE_WAIT;
	MsgOK:=FALSE;
	MsgCancel:=FALSE;
	SFCRun:=FALSE;
END_IF
END_ACTION

ACTION OpenSeperatorWender_action:
ST03_464_Y71_0.MoveInit:=TRUE;		(* Förderband  Zuführung Vereinzelner Wender AST/GST *)
END_ACTION

ACTION WaitForPart__entry:
ProcessMessage01:='';
Delay.IN:=FALSE;
Delay();
END_ACTION

ACTION WaitForPart__action:
ProcessMessage01:='1IM6';(*'warte auf Teil in Vereinzelung*)
Delay.IN:=ST03_462_B70_0.BitInToCheck; 		 (* Züführung  ISK auf Übergabeposition Roboter Palettierer  *)
Delay.PT:=T#800ms;
Delay();
END_ACTION

ACTION WaitForPart__exit:
ProcessMessage01:='';
END_ACTION

ACTION CloseSeperatorWender_action:
ST03_464_Y71_0.MoveWork:=TRUE;		(* Förderband  Zuführung Vereinzelner Wender AST/GST *)
END_ACTION

ACTION ZylVakuumWork_action:
ST03_464_Y71_1.MoveWork:=TRUE;		(*  Förderband  Zuführung Zylinder Vakuumdüsen AST/GST*)
END_ACTION

ACTION VakuumOn_action:
ST03_464_Y71_5.MoveWork:=TRUE;	(*  Förderband  Vakuumdüsen EIN/AUS *)
END_ACTION

ACTION WenderWork_action:
ST03_464_Y71_2.MoveWork:=TRUE;		(* Förderband  Zuführung Wender Einlauf / Auslauf *)
END_ACTION

ACTION ZylVakuumInit__action:
ST03_464_Y71_1.MoveInit:=TRUE;		(*  Förderband  Zuführung Zylinder Vakuumdüsen AST/GST*)
END_ACTION

ACTION VakuumOff__action:
ST03_464_Y71_5.MoveInit:=TRUE;	(*  Förderband  Vakuumdüsen EIN/AUS *)
END_ACTION

ACTION Delay__entry:
Delay(IN:=FALSE);
END_ACTION

ACTION Delay__action:
Delay(IN:=TRUE,PT:=t#2000ms);
END_ACTION

ACTION Delay__exit:
Delay(IN:=FALSE);
END_ACTION

ACTION WenderInit_entry:
Delay(IN:=FALSE);
END_ACTION

ACTION WenderInit_action:
ST03_464_Y71_2.MoveInit:=TRUE;		(* Förderband  Zuführung Wender Einlauf / Auslauf *)
END_ACTION

ACTION VakuumNOK_entry:
MessageHandler.ClearMessageLines(sVisu:=Visu.Message);
END_ACTION

ACTION VakuumNOK_action:
MessageHandler.Msg.ID:='PM119';
MessageHandler.Msg.Name:='Vakuum nicht OK';
MessageHandler.Msg.Text:='ST03 Vakuum an der Wendestation nicht OK';
MessageHandler.Msg.Color:=Color.red;
MessageHandler.Msg.Station:=1;


MessageHandler(
	Prio:=2, 							(*1=highest, .. , 4=lowest*)
	Btn1Addr:=ADR(MsgOk),			(*Address of Button1 , if Zero then Button is unvisible*)
	Btn2Addr:=ADR(MsgCancel),			(*Address of Button2 , if Zero then Button is unvisible*)
	sVisu:=Visu.Message);
END_ACTION

ACTION VakuumNOK_exit:
MsgOk:=FALSE;
MsgCancel:=FALSE;
END_ACTION

ACTION ZylVakuumInit_action:
ST03_464_Y71_1.MoveInit:=TRUE;		(*  Förderband  Zuführung Zylinder Vakuumdüsen AST/GST*)
END_ACTION

ACTION VakuumOff_action:
ST03_464_Y71_5.MoveInit:=TRUE;	(*  Förderband  Vakuumdüsen EIN/AUS *)
END_ACTION

ACTION SeqEnd2_entry:
WenderDone:=TRUE;
END_ACTION

ACTION SeqEnd2_exit:
WenderDone:=FALSE;
END_ACTION

TRANSITION WenderPosEmptyr:
NOT ST03_462_B70_0.BitInToCheck AND	(*Förderband  ISK anwesend Wender*)
NOT  ST03_464_B71_7.BitInToCheck	 AND	(*Förderband   Staustrecke mitte voll*)
ST03_463_B70_5.ValveSensor				(* Züführung  ISK Wendestation Einlauf GST*)
END_TRANSITION

TRANSITION StateOK:
ST03_464_Y71_0.State = STATE_OK 	(* Förderband  Zuführung Vereinzelner Wender AST/GST *)
END_TRANSITION

TRANSITION WenderPosFulll:
ST03_462_B70_0.BitInToCheck AND	(*Förderband  ISK anwesend Wender*)
NOT  ST03_464_B71_7.BitInToCheck  AND	(*Förderband   Staustrecke mitte voll*)
ST03_463_B70_5.ValveSensor				(* Züführung  ISK Wendestation Einlauf GST*)
END_TRANSITION

TRANSITION Part Ready:
Delay.Q
END_TRANSITION

TRANSITION StateOK:
ST03_464_Y71_0.State = STATE_OK AND	(* Förderband  Zuführung Vereinzelner Wender AST/GST *)
ST03_464_Y71_1.State = STATE_OK	AND	(*   Förderband  Zuführung Zylinder Vakuumdüsen AST/GST *)
ST03_464_Y71_5.State = STATE_OK		(*  Förderband  Vakuumdüsen EIN/AUS *)
END_TRANSITION

TRANSITION CheckVakuum:
ST03_464_B71_6.BitInToCheck	(*Förderband  Vakuum vorhanden*)
END_TRANSITION

TRANSITION StateOK:
ST03_464_Y71_2.State = STATE_OK 	(* Förderband  ZuführungWender Einlauf / Auslauf  *)
END_TRANSITION

TRANSITION StateOK:
ST03_464_Y71_1.State = STATE_OK	AND	(*   Förderband  Zuführung Zylinder Vakuumdüsen AST/GST *)
ST03_464_Y71_5.State = STATE_OK		(*  Förderband  Vakuumdüsen EIN/AUS *)
END_TRANSITION

TRANSITION CheckSens:
ST03_464_B71_7.BitInToCheck	(* Förderband   Staustrecke mitte vol*) OR
delay.Q
END_TRANSITION

TRANSITION StateOK:
ST03_464_Y71_2.State = STATE_OK 	(* Förderband  ZuführungWender Einlauf / Auslauf  *)
END_TRANSITION

TRANSITION StateOK:
ST03_464_Y71_1.State = STATE_OK	AND	(*   Förderband  Zuführung Zylinder Vakuumdüsen AST/GST *)
ST03_464_Y71_5.State = STATE_OK		(*  Förderband  Vakuumdüsen EIN/AUS *)
END_TRANSITION
END_PROGRAM

(* POU Stations/ST_03_Ruestsaetze/ST_03_SFCs/Zufuehrungen/ST03_NOX_4pol_Zufuehrung, SFC *)
 PROGRAM ST03_NOX_4pol_Zufuehrung
VAR_OUTPUT
	SFCCurrentPOU		: STRING:='ST03_NOX_4pol_Zufuehrung';
	SFCCurrentStep		: STRING:='';
	FB_CurrentStepHistorie:FB_CurrentStepHistorie;
	SFCTime			: DINT;
	State   				: StateObject	:= STATE_WAIT;
	Result  				: StateResult;
END_VAR
VAR_INPUT
	Start					:BOOL;
END_VAR
VAR
	MsgOK				: BOOL;
	MsgCancel			: BOOL;
	SFCRun				: BOOL;
	SFCTimeStart		: TIME;
	Delay				: TON;
	(* Userdefinded area *)

END_VAR
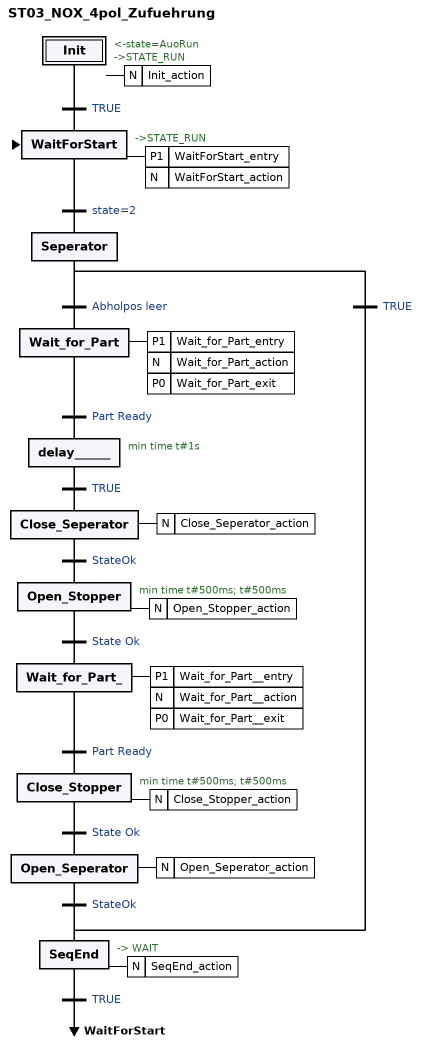
INITIAL_STEP Init: (* <-state=AuoRun / ->STATE_RUN *)
	Init_action(N);
END_STEP
TRANSITION FROM Init TO WaitForStart := TRUE;
END_TRANSITION
STEP WaitForStart: (* ->STATE_RUN *)
	WaitForStart_entry(P1);
	WaitForStart_action(N);
END_STEP
TRANSITION FROM WaitForStart TO Seperator := state=2;
END_TRANSITION
STEP Seperator:
END_STEP
TRANSITION FROM Seperator TO Wait_for_Part := Abholpos leer;
END_TRANSITION
TRANSITION FROM Seperator TO SeqEnd := TRUE;
END_TRANSITION
STEP Wait_for_Part:
	Wait_for_Part_entry(P1);
	Wait_for_Part_action(N);
	Wait_for_Part_exit(P0);
END_STEP
TRANSITION FROM Wait_for_Part TO delay______ := Part Ready;
END_TRANSITION
STEP delay______: (* min time t#1s *)
END_STEP
TRANSITION FROM delay______ TO Close_Seperator := TRUE;
END_TRANSITION
STEP Close_Seperator:
	Close_Seperator_action(N);
END_STEP
TRANSITION FROM Close_Seperator TO Open_Stopper := StateOk;
END_TRANSITION
STEP Open_Stopper: (* min time t#500ms; t#500ms *)
	Open_Stopper_action(N);
END_STEP
TRANSITION FROM Open_Stopper TO Wait_for_Part_ := State Ok;
END_TRANSITION
STEP Wait_for_Part_:
	Wait_for_Part__entry(P1);
	Wait_for_Part__action(N);
	Wait_for_Part__exit(P0);
END_STEP
TRANSITION FROM Wait_for_Part_ TO Close_Stopper := Part Ready;
END_TRANSITION
STEP Close_Stopper: (* min time t#500ms; t#500ms *)
	Close_Stopper_action(N);
END_STEP
TRANSITION FROM Close_Stopper TO Open_Seperator := State Ok;
END_TRANSITION
STEP Open_Seperator:
	Open_Seperator_action(N);
END_STEP
TRANSITION FROM Open_Seperator TO SeqEnd := StateOk;
END_TRANSITION
STEP SeqEnd: (* -> WAIT *)
	SeqEnd_action(N);
END_STEP
TRANSITION FROM SeqEnd TO WaitForStart := TRUE;
END_TRANSITION

ACTION Init_action:
Start:=FALSE;
State:=STATE_WAIT;
MsgOK:=FALSE;
MsgCancel:=FALSE;
SFCRun:=FALSE;
Result:=RESULT_NON;
END_ACTION

ACTION WaitForStart_entry:
;
END_ACTION

ACTION WaitForStart_action:
IF 	Start   THEN
	State:=STATE_RUN;
	Result:=RESULT_NON;
	SFCTimeStart:=TIME();
	Start:=FALSE;
ELSE
	State:=STATE_WAIT;
	MsgOK:=FALSE;
	MsgCancel:=FALSE;
	SFCRun:=FALSE;
END_IF
END_ACTION

ACTION Wait_for_Part_entry:
ProcessMessage01:='';
Delay.IN:=FALSE;
Delay();
END_ACTION

ACTION Wait_for_Part_action:
ProcessMessage01:='1IM9';(*warte auf Teil in Stopper*)
Delay.IN:=ST03_491_B69_5.BitInToCheck; 		(*  ISK an stopper.*)
Delay.PT:=T#500ms;
Delay();
END_ACTION

ACTION Wait_for_Part_exit:
ProcessMessage01:='';
END_ACTION

ACTION Close_Seperator_action:
ST03_492_Y70_0.MoveWork:=TRUE;		(* Förderband  Zuführung Vereinzler AST/GST *)
END_ACTION

ACTION Open_Stopper_action:
ST03_492_Y70_1.MoveWork:=TRUE;		(* Förderband  Züführung Stopper AST/GST *)
END_ACTION

ACTION Wait_for_Part__entry:
ProcessMessage01:='';
Delay.IN:=FALSE;
Delay();
END_ACTION

ACTION Wait_for_Part__action:
ProcessMessage01:='1IM10';(*warte auf Teil in Abholposition*)
Delay.IN:=ST03_491_B69_7.BitInToCheck; 		 (* Schnittstelle Iso auf Übergabeposition Roboter *)
Delay.PT:=T#500ms;
Delay();
END_ACTION

ACTION Wait_for_Part__exit:
ProcessMessage01:='';
END_ACTION

ACTION Close_Stopper_action:
ST03_492_Y70_1.MoveInit:=TRUE;		(* Förderband  Züführung Stopper AST/GST *)
END_ACTION

ACTION Open_Seperator_action:
ST03_492_Y70_0.MoveInit:=TRUE;		(* Förderband  Zuführung Vereinzler AST/GST *)
END_ACTION

ACTION SeqEnd_action:
SFCTime:=TIME_TO_DINT(TIME()-SFCTimeStart);
State:=STATE_WAIT;
END_ACTION

TRANSITION Abholpos leer:
NOT  ST03_491_B69_7.BitInToCheck		(*  ISK auf Abholposition Robi*)
END_TRANSITION

TRANSITION Part Ready:
Delay.Q AND
NOT ST03_491_B69_7.BitInToCheck	AND		(*  ISK auf Abholposition Robi*)
ST03_491_B69_5.BitInToCheck	AND				(*  ISK anwesend am Stoper*)
Robot01.ActualArea <> 4
END_TRANSITION

TRANSITION StateOk:
ST03_492_Y70_0.State=STATE_OK 	(* Förderband  Zuführung Vereinzler AST/GST *)
END_TRANSITION

TRANSITION State Ok:
ST03_492_Y70_1.State=STATE_OK 	(* Förderband  Züführung Stopper AST/GST *)
END_TRANSITION

TRANSITION Part Ready:
Delay.Q AND
Robot01.ActualArea <> 4
END_TRANSITION

TRANSITION State Ok:
ST03_492_Y70_1.State=STATE_OK 	(* Förderband  Züführung Stopper AST/GST *)
END_TRANSITION

TRANSITION StateOk:
ST03_492_Y70_0.State=STATE_OK 	(* Förderband  Zuführung Vereinzler AST/GST *)
END_TRANSITION
END_PROGRAM

(* POU Stations/ST_03_Ruestsaetze/ST_03_SFCs/Zufuehrungen/ST03_88pol_Zufuehrung, SFC *)
 PROGRAM ST03_88pol_Zufuehrung
VAR_OUTPUT
	SFCCurrentPOU			: STRING:='ST03_88pol_Zufuehrung';
	SFCCurrentStep			: STRING:='';
	FB_CurrentStepHistorie:FB_CurrentStepHistorie;
	SFCTime					: DINT;
	State   				: StateObject	:= STATE_WAIT;
	Result  				: StateResult;
END_VAR
VAR_INPUT
	Start					:BOOL;
END_VAR
VAR
	MsgOK				: BOOL;
	MsgCancel			: BOOL;
	SFCRun				: BOOL;
	SFCTimeStart		: TIME;
	Delay				: TON;
	(* Userdefinded area *)

END_VAR
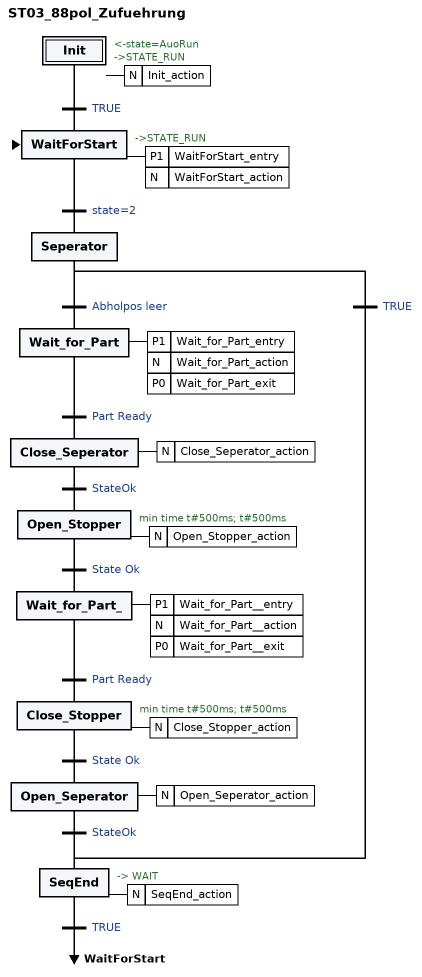
INITIAL_STEP Init: (* <-state=AuoRun / ->STATE_RUN *)
	Init_action(N);
END_STEP
TRANSITION FROM Init TO WaitForStart := TRUE;
END_TRANSITION
STEP WaitForStart: (* ->STATE_RUN *)
	WaitForStart_entry(P1);
	WaitForStart_action(N);
END_STEP
TRANSITION FROM WaitForStart TO Seperator := state=2;
END_TRANSITION
STEP Seperator:
END_STEP
TRANSITION FROM Seperator TO Wait_for_Part := Abholpos leer;
END_TRANSITION
TRANSITION FROM Seperator TO SeqEnd := TRUE;
END_TRANSITION
STEP Wait_for_Part:
	Wait_for_Part_entry(P1);
	Wait_for_Part_action(N);
	Wait_for_Part_exit(P0);
END_STEP
TRANSITION FROM Wait_for_Part TO Close_Seperator := Part Ready;
END_TRANSITION
STEP Close_Seperator:
	Close_Seperator_action(N);
END_STEP
TRANSITION FROM Close_Seperator TO Open_Stopper := StateOk;
END_TRANSITION
STEP Open_Stopper: (* min time t#500ms; t#500ms *)
	Open_Stopper_action(N);
END_STEP
TRANSITION FROM Open_Stopper TO Wait_for_Part_ := State Ok;
END_TRANSITION
STEP Wait_for_Part_:
	Wait_for_Part__entry(P1);
	Wait_for_Part__action(N);
	Wait_for_Part__exit(P0);
END_STEP
TRANSITION FROM Wait_for_Part_ TO Close_Stopper := Part Ready;
END_TRANSITION
STEP Close_Stopper: (* min time t#500ms; t#500ms *)
	Close_Stopper_action(N);
END_STEP
TRANSITION FROM Close_Stopper TO Open_Seperator := State Ok;
END_TRANSITION
STEP Open_Seperator:
	Open_Seperator_action(N);
END_STEP
TRANSITION FROM Open_Seperator TO SeqEnd := StateOk;
END_TRANSITION
STEP SeqEnd: (* -> WAIT *)
	SeqEnd_action(N);
END_STEP
TRANSITION FROM SeqEnd TO WaitForStart := TRUE;
END_TRANSITION

ACTION Init_action:
Start:=FALSE;
State:=STATE_WAIT;
MsgOK:=FALSE;
MsgCancel:=FALSE;
SFCRun:=FALSE;
Result:=RESULT_NON;
END_ACTION

ACTION WaitForStart_entry:
State:=STATE_OK;
END_ACTION

ACTION WaitForStart_action:
IF 	Start   THEN
	State:=STATE_RUN;
	Result:=RESULT_NON;
	SFCTimeStart:=TIME();
	Start:=FALSE;
ELSE
	State:=STATE_WAIT;
	MsgOK:=FALSE;
	MsgCancel:=FALSE;
	SFCRun:=FALSE;
END_IF
END_ACTION

ACTION Wait_for_Part_entry:
ProcessMessage01:='';
Delay.IN:=FALSE;
Delay();
END_ACTION

ACTION Wait_for_Part_action:
State:=STATE_RUN;
ProcessMessage01:='1IM9';(*warte auf Teil in Stopper*)
Delay.IN:=ST03_501_B69_6.BitInToCheck; 		(*  ISK an stopper.*)
Delay.PT:=T#500ms;
Delay();
END_ACTION

ACTION Wait_for_Part_exit:
ProcessMessage01:='';
END_ACTION

ACTION Close_Seperator_action:
ST03_502_Y70_1.MoveWork:=TRUE;		(* Förderband  Zuführung Vereinzler AST/GST *)
END_ACTION

ACTION Open_Stopper_action:
ST03_502_Y70_2.MoveWork:=TRUE;		(* Förderband  Züführung Stopper AST/GST *)
END_ACTION

ACTION Wait_for_Part__entry:
ProcessMessage01:='';
Delay.IN:=FALSE;
Delay();
END_ACTION

ACTION Wait_for_Part__action:
ProcessMessage01:='1IM10';(*warte auf Teil in Abholposition*)
Delay.IN:=ST03_501_B69_7.BitInToCheck; 		 (* ISK auf Abholposition Robi *)
Delay.PT:=T#500ms;
Delay();
END_ACTION

ACTION Wait_for_Part__exit:
ProcessMessage01:='';
END_ACTION

ACTION Close_Stopper_action:
ST03_502_Y70_2.MoveInit:=TRUE;		(* Förderband  Züführung Stopper AST/GST *)
END_ACTION

ACTION Open_Seperator_action:
ST03_502_Y70_1.MoveInit:=TRUE;		(* Förderband  Zuführung Vereinzler AST/GST *)
END_ACTION

ACTION SeqEnd_action:
SFCTime:=TIME_TO_DINT(TIME()-SFCTimeStart);
State:=STATE_WAIT;
END_ACTION

TRANSITION Abholpos leer:
NOT  ST03_501_B69_7.BitInToCheck		(*  ISK auf Abholposition Robi*)
END_TRANSITION

TRANSITION Part Ready:
Delay.Q AND
NOT ST03_501_B69_7.BitInToCheck	AND		(*  ISK auf Abholposition Robi*)
ST03_501_B69_6.BitInToCheck	AND				(*  ISK anwesend am Stoper*)
Robot01.ActualArea <> 4
END_TRANSITION

TRANSITION StateOk:
ST03_502_Y70_1.State=STATE_OK 	(* Förderband  Zuführung Vereinzler AST/GST *)
END_TRANSITION

TRANSITION State Ok:
ST03_502_Y70_2.State=STATE_OK 	(* Förderband  Züführung Stopper AST/GST *)
END_TRANSITION

TRANSITION Part Ready:
Delay.Q AND
Robot01.ActualArea <> 4
END_TRANSITION

TRANSITION State Ok:
ST03_502_Y70_2.State=STATE_OK 	(* Förderband  Züführung Stopper AST/GST *)
END_TRANSITION

TRANSITION StateOk:
ST03_502_Y70_1.State=STATE_OK 	(* Förderband  Zuführung Vereinzler AST/GST *)
END_TRANSITION
END_PROGRAM

(* POU Stations/ST_03_Ruestsaetze/ST_03_SFCs/Zufuehrungen/ST03_7pol_Zufuehrung, SFC *)
 PROGRAM ST03_7pol_Zufuehrung
VAR_OUTPUT
	SFCCurrentPOU			: STRING:='ST03_7pol_Zufuehrung';
	SFCCurrentStep			: STRING:='';
	FB_CurrentStepHistorie	:FB_CurrentStepHistorie;
	SFCTime					: DINT;
	State   				: StateObject	:= STATE_WAIT;
	Result  				: StateResult;
END_VAR
VAR_INPUT
	Start					:BOOL;
END_VAR
VAR
	MsgOK				: BOOL;
	MsgCancel			: BOOL;
	SFCRun			: BOOL;
	SFCTimeStart		: TIME;
	Delay				: TON;
	Delay2				: TON;
	(* Userdefinded area *)

END_VAR
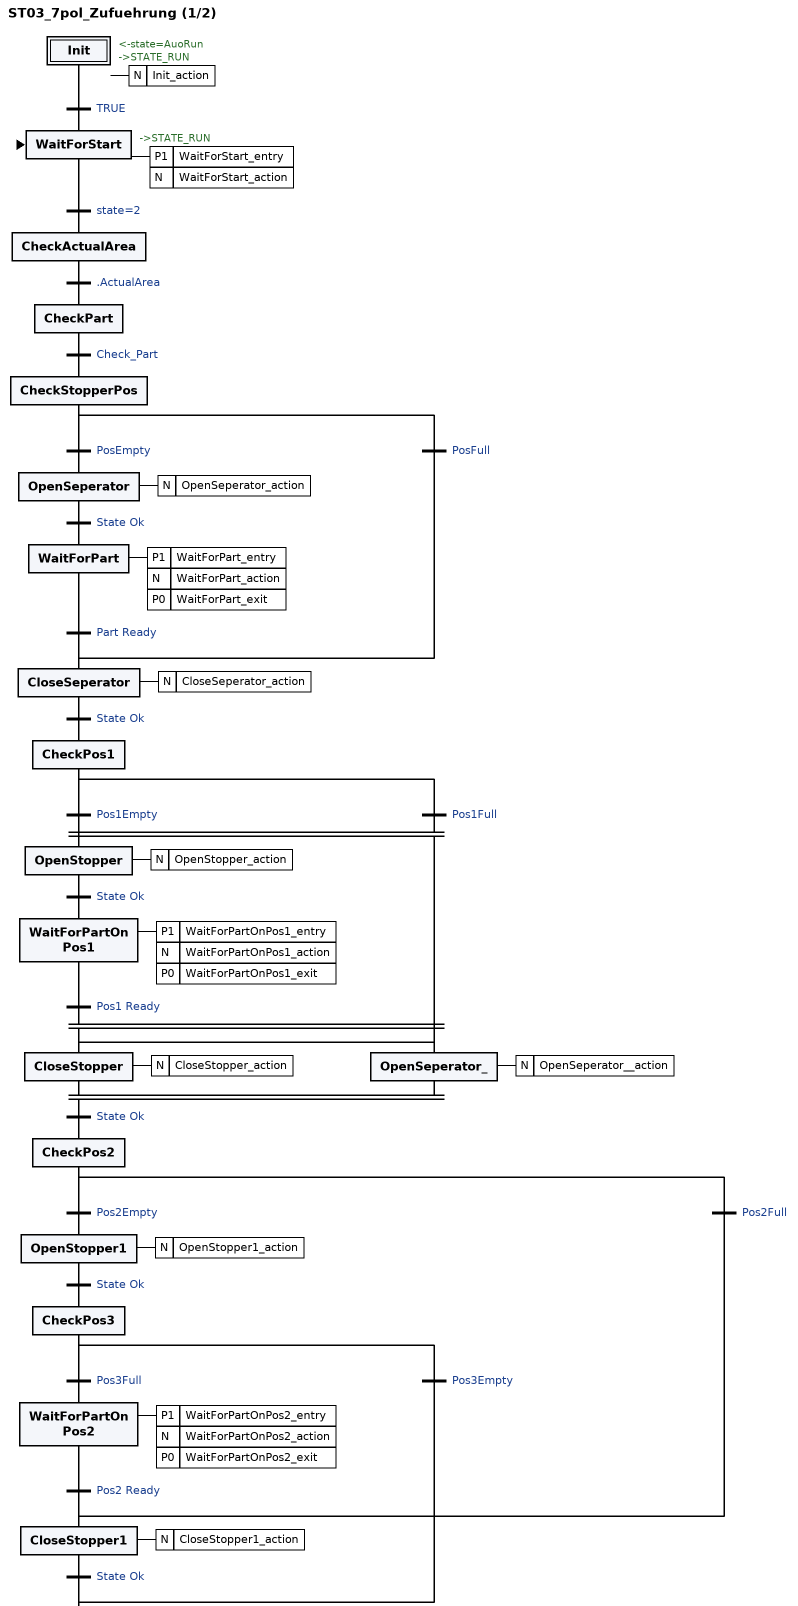
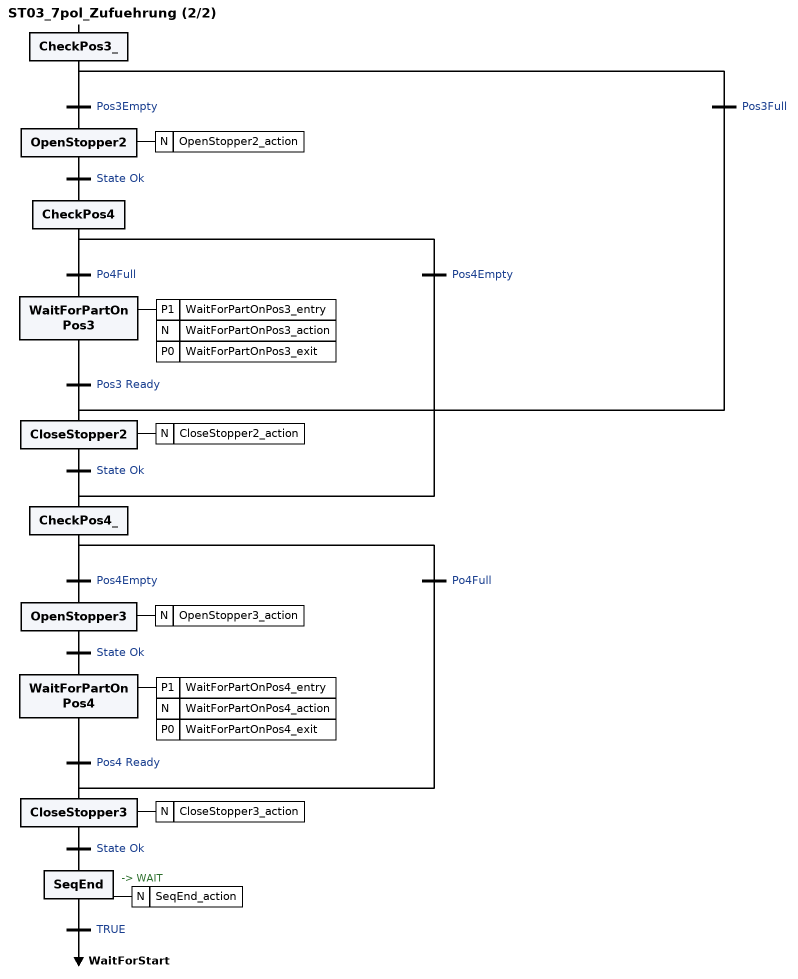
INITIAL_STEP Init: (* <-state=AuoRun / ->STATE_RUN *)
	Init_action(N);
END_STEP
TRANSITION FROM Init TO WaitForStart := TRUE;
END_TRANSITION
STEP WaitForStart: (* ->STATE_RUN *)
	WaitForStart_entry(P1);
	WaitForStart_action(N);
END_STEP
TRANSITION FROM WaitForStart TO CheckActualArea := state=2;
END_TRANSITION
STEP CheckActualArea:
END_STEP
TRANSITION FROM CheckActualArea TO CheckPart := .ActualArea;
END_TRANSITION
STEP CheckPart:
END_STEP
TRANSITION FROM CheckPart TO CheckStopperPos := Check_Part;
END_TRANSITION
STEP CheckStopperPos:
END_STEP
TRANSITION FROM CheckStopperPos TO OpenSeperator := PosEmpty;
END_TRANSITION
TRANSITION FROM CheckStopperPos TO CloseSeperator := PosFull;
END_TRANSITION
STEP OpenSeperator:
	OpenSeperator_action(N);
END_STEP
TRANSITION FROM OpenSeperator TO WaitForPart := State Ok;
END_TRANSITION
STEP WaitForPart:
	WaitForPart_entry(P1);
	WaitForPart_action(N);
	WaitForPart_exit(P0);
END_STEP
TRANSITION FROM WaitForPart TO CloseSeperator := Part Ready;
END_TRANSITION
STEP CloseSeperator:
	CloseSeperator_action(N);
END_STEP
TRANSITION FROM CloseSeperator TO CheckPos1 := State Ok;
END_TRANSITION
STEP CheckPos1:
END_STEP
TRANSITION FROM CheckPos1 TO OpenStopper := Pos1Empty;
END_TRANSITION
TRANSITION FROM CheckPos1 TO (CloseStopper, OpenSeperator_) := Pos1Full;
END_TRANSITION
STEP OpenStopper:
	OpenStopper_action(N);
END_STEP
TRANSITION FROM OpenStopper TO WaitForPartOnPos1 := State Ok;
END_TRANSITION
STEP WaitForPartOnPos1:
	WaitForPartOnPos1_entry(P1);
	WaitForPartOnPos1_action(N);
	WaitForPartOnPos1_exit(P0);
END_STEP
TRANSITION FROM WaitForPartOnPos1 TO (CloseStopper, OpenSeperator_) := Pos1 Ready;
END_TRANSITION
STEP CloseStopper:
	CloseStopper_action(N);
END_STEP
STEP OpenSeperator_:
	OpenSeperator__action(N);
END_STEP
TRANSITION FROM (CloseStopper, OpenSeperator_) TO CheckPos2 := State Ok;
END_TRANSITION
STEP CheckPos2:
END_STEP
TRANSITION FROM CheckPos2 TO OpenStopper1 := Pos2Empty;
END_TRANSITION
TRANSITION FROM CheckPos2 TO CloseStopper1 := Pos2Full;
END_TRANSITION
STEP OpenStopper1:
	OpenStopper1_action(N);
END_STEP
TRANSITION FROM OpenStopper1 TO CheckPos3 := State Ok;
END_TRANSITION
STEP CheckPos3:
END_STEP
TRANSITION FROM CheckPos3 TO WaitForPartOnPos2 := Pos3Full;
END_TRANSITION
TRANSITION FROM CheckPos3 TO CheckPos3_ := Pos3Empty;
END_TRANSITION
STEP WaitForPartOnPos2:
	WaitForPartOnPos2_entry(P1);
	WaitForPartOnPos2_action(N);
	WaitForPartOnPos2_exit(P0);
END_STEP
TRANSITION FROM WaitForPartOnPos2 TO CloseStopper1 := Pos2 Ready;
END_TRANSITION
STEP CloseStopper1:
	CloseStopper1_action(N);
END_STEP
TRANSITION FROM CloseStopper1 TO CheckPos3_ := State Ok;
END_TRANSITION
STEP CheckPos3_:
END_STEP
TRANSITION FROM CheckPos3_ TO OpenStopper2 := Pos3Empty;
END_TRANSITION
TRANSITION FROM CheckPos3_ TO CloseStopper2 := Pos3Full;
END_TRANSITION
STEP OpenStopper2:
	OpenStopper2_action(N);
END_STEP
TRANSITION FROM OpenStopper2 TO CheckPos4 := State Ok;
END_TRANSITION
STEP CheckPos4:
END_STEP
TRANSITION FROM CheckPos4 TO WaitForPartOnPos3 := Po4Full;
END_TRANSITION
TRANSITION FROM CheckPos4 TO CheckPos4_ := Pos4Empty;
END_TRANSITION
STEP WaitForPartOnPos3:
	WaitForPartOnPos3_entry(P1);
	WaitForPartOnPos3_action(N);
	WaitForPartOnPos3_exit(P0);
END_STEP
TRANSITION FROM WaitForPartOnPos3 TO CloseStopper2 := Pos3 Ready;
END_TRANSITION
STEP CloseStopper2:
	CloseStopper2_action(N);
END_STEP
TRANSITION FROM CloseStopper2 TO CheckPos4_ := State Ok;
END_TRANSITION
STEP CheckPos4_:
END_STEP
TRANSITION FROM CheckPos4_ TO OpenStopper3 := Pos4Empty;
END_TRANSITION
TRANSITION FROM CheckPos4_ TO CloseStopper3 := Po4Full;
END_TRANSITION
STEP OpenStopper3:
	OpenStopper3_action(N);
END_STEP
TRANSITION FROM OpenStopper3 TO WaitForPartOnPos4 := State Ok;
END_TRANSITION
STEP WaitForPartOnPos4:
	WaitForPartOnPos4_entry(P1);
	WaitForPartOnPos4_action(N);
	WaitForPartOnPos4_exit(P0);
END_STEP
TRANSITION FROM WaitForPartOnPos4 TO CloseStopper3 := Pos4 Ready;
END_TRANSITION
STEP CloseStopper3:
	CloseStopper3_action(N);
END_STEP
TRANSITION FROM CloseStopper3 TO SeqEnd := State Ok;
END_TRANSITION
STEP SeqEnd: (* -> WAIT *)
	SeqEnd_action(N);
END_STEP
TRANSITION FROM SeqEnd TO WaitForStart := TRUE;
END_TRANSITION

ACTION Init_action:
Start:=FALSE;
State:=STATE_WAIT;
MsgOK:=FALSE;
MsgCancel:=FALSE;
SFCRun:=FALSE;
Result:=RESULT_NON;
END_ACTION

ACTION WaitForStart_entry:
;
END_ACTION

ACTION WaitForStart_action:
IF 	Start   THEN
	State:=STATE_RUN;
	Result:=RESULT_NON;
	SFCTimeStart:=TIME();
	Start:=FALSE;
ELSE
	State:=STATE_WAIT;
	MsgOK:=FALSE;
	MsgCancel:=FALSE;
	SFCRun:=FALSE;
END_IF
END_ACTION

ACTION OpenSeperator_action:
ST03_515_Y72_2.MoveInit:=TRUE;		(* Führungsschiene  Zuführung Vereinzler AST/GST *)
END_ACTION

ACTION WaitForPart_entry:
ProcessMessage02:='';
Delay(IN:=FALSE);
END_ACTION

ACTION WaitForPart_action:
ProcessMessage02:='2IM6';						(*warte auf Teil Übergabeposition 1*)
END_ACTION

ACTION WaitForPart_exit:
ProcessMessage02:='';
END_ACTION

ACTION CloseSeperator_action:
ST03_515_Y72_2.MoveWork:=TRUE;		(* Führungsschiene  Zuführung Vereinzler AST/GST *)
END_ACTION

ACTION OpenStopper_action:
ST03_515_Y72_3.MoveWork:=TRUE;		(* Führungsschiene  Zuführung Stopper AST/GST *)
END_ACTION

ACTION WaitForPartOnPos1_entry:
ProcessMessage02:='';
Delay(IN:=FALSE);
END_ACTION

ACTION WaitForPartOnPos1_action:
ProcessMessage02:='2IM6';						(*warte auf Teil Übergabeposition 1*)
END_ACTION

ACTION WaitForPartOnPos1_exit:
ProcessMessage02:='';
END_ACTION

ACTION CloseStopper_action:
ST03_515_Y72_3.MoveInit:=TRUE;		(* Führungsschiene  Zuführung Stopper AST/GST *)
END_ACTION

ACTION OpenSeperator__action:
ST03_515_Y72_2.MoveInit:=TRUE;		(* Führungsschiene  Zuführung Vereinzler AST/GST *)
END_ACTION

ACTION OpenStopper1_action:
ST03_515_Y72_4.MoveWork:=TRUE;		(* Übergabeposition Stopper 1 *)
END_ACTION

ACTION WaitForPartOnPos2_entry:
ProcessMessage02:='';
Delay(IN:=FALSE);
END_ACTION

ACTION WaitForPartOnPos2_action:
ProcessMessage02:='2IM5';						(*warte auf Teil Übergabeposition 2*)
END_ACTION

ACTION WaitForPartOnPos2_exit:
ProcessMessage02:='';
END_ACTION

ACTION CloseStopper1_action:
ST03_515_Y72_4.MoveInit:=TRUE;		(* Übergabeposition Stopper 1 *)
END_ACTION

ACTION OpenStopper2_action:
ST03_515_Y72_5.MoveWork:=TRUE;		(* Übergabeposition Stopper 2 *)
END_ACTION

ACTION WaitForPartOnPos3_entry:
ProcessMessage02:='';
Delay(IN:=FALSE);
END_ACTION

ACTION WaitForPartOnPos3_action:
ProcessMessage02:='2IM4';						(*warte auf Teil Übergabeposition 3*)
END_ACTION

ACTION WaitForPartOnPos3_exit:
ProcessMessage02:='';
END_ACTION

ACTION CloseStopper2_action:
ST03_515_Y72_5.MoveInit:=TRUE;		(* Übergabeposition Stopper 2 *)
END_ACTION

ACTION OpenStopper3_action:
ST03_515_Y72_6.MoveWork:=TRUE;		(* Übergabeposition Stopper 3 *)
END_ACTION

ACTION WaitForPartOnPos4_entry:
ProcessMessage02:='';
Delay(IN:=FALSE);
END_ACTION

ACTION WaitForPartOnPos4_action:
ProcessMessage02:='2IM3';						(*warte auf Teil Übergabeposition 4*)
Delay(
	IN:=NOT ST03_513_B70_7.BitInToCheck AND	(* ISK auf Übergabeposition  1*)
		NOT ST03_514_B71_2.BitInToCheck AND	(* ISK auf Übergabeposition  2*)
		NOT ST03_514_B71_5.BitInToCheck AND	(* ISK auf Übergabeposition  3*)
		NOT ST03_514_B71_6.BitInToCheck		(* ISK auf Übergabeposition  4*),
	PT:=t#1s);
END_ACTION

ACTION WaitForPartOnPos4_exit:
ProcessMessage02:='';
Delay(IN:=FALSE);
END_ACTION

ACTION CloseStopper3_action:
ST03_515_Y72_6.MoveInit:=TRUE;		(* Übergabeposition Stopper 3 *)
END_ACTION

ACTION SeqEnd_action:
SFCTime:=TIME_TO_DINT(TIME()-SFCTimeStart);
State:=STATE_WAIT;
END_ACTION

TRANSITION .ActualArea:
Robot01.ActualArea <> 4
END_TRANSITION

TRANSITION Check_Part:
NOT ST03_513_B70_7.BitInToCheck OR	(* ISK auf Übergabeposition  1*)
NOT ST03_514_B71_2.BitInToCheck OR	(* ISK auf Übergabeposition  2*)
NOT ST03_514_B71_5.BitInToCheck OR	(* ISK auf Übergabeposition  3*)
NOT ST03_514_B71_6.BitInToCheck		(* ISK auf Übergabeposition  4*)
END_TRANSITION

TRANSITION PosEmpty:
NOT ST03_513_B70_4.BitInToCheck			 	(*  ISK anwesend am Stopper*)
END_TRANSITION

TRANSITION State Ok:
ST03_515_Y72_2.State=STATE_OK (* Führungsschiene  Zuführung Vereinzler AST/GST *)
END_TRANSITION

TRANSITION Part Ready:
ST03_513_B70_4.BitInToCheck	(*  ISK anwesend am Stopper*)
END_TRANSITION

TRANSITION PosFull:
ST03_513_B70_4.BitInToCheck			 	(*  ISK anwesend am Stopper*)
END_TRANSITION

TRANSITION State Ok:
ST03_515_Y72_2.State=STATE_OK (* Führungsschiene  Zuführung Vereinzler AST/GST *)
END_TRANSITION

TRANSITION Pos1Empty:
NOT ST03_513_B70_7.BitInToCheck AND 	(*  ISK auf Übergabeposition 1*)
Robot01.ActualArea <> 4
END_TRANSITION

TRANSITION State Ok:
ST03_515_Y72_3.State=STATE_OK 	(* Führungsschiene  Zuführung Stopper AST/GST *)
END_TRANSITION

TRANSITION Pos1 Ready:
ST03_513_B70_7.BitInToCheck 		 (* ISK auf Übergabeposition 1 *)
END_TRANSITION

TRANSITION Pos1Full:
ST03_513_B70_7.BitInToCheck 	(*  ISK auf Übergabeposition 1*)
END_TRANSITION

TRANSITION State Ok:
ST03_515_Y72_3.State=STATE_OK AND 	(* Führungsschiene  Zuführung Stopper AST/GST *)
ST03_515_Y72_2.State=STATE_OK (* Führungsschiene  Zuführung Vereinzler AST/GST *)
END_TRANSITION

TRANSITION Pos2Empty:
NOT ST03_514_B71_2.BitInToCheck  	(*  ISK auf Übergabeposition 2*)
END_TRANSITION

TRANSITION State Ok:
ST03_515_Y72_4.State=STATE_OK 	(* Übergabeposition Stopper 1 AST/GST *)
END_TRANSITION

TRANSITION Pos3Full:
ST03_514_B71_5.BitInToCheck	 	(*  ISK auf Übergabeposition 3*)
END_TRANSITION

TRANSITION Pos3Empty:
NOT ST03_514_B71_5.BitInToCheck  	(*  ISK auf Übergabeposition 3*)
END_TRANSITION

TRANSITION Pos2 Ready:
ST03_514_B71_2.BitInToCheck 		 (* ISK auf Übergabeposition 2 *)
END_TRANSITION

TRANSITION Pos2Full:
ST03_514_B71_2.BitInToCheck	 	(*  ISK auf Übergabeposition 2*)
END_TRANSITION

TRANSITION State Ok:
ST03_515_Y72_4.State=STATE_OK 	(* Übergabeposition Stopper 1 AST/GST *)
END_TRANSITION

TRANSITION Pos3Empty:
NOT ST03_514_B71_5.BitInToCheck  	(*  ISK auf Übergabeposition 3*)
END_TRANSITION

TRANSITION State Ok:
ST03_515_Y72_5.State=STATE_OK 	(* Übergabeposition Stopper 2 AST/GST *)
END_TRANSITION

TRANSITION Po4Full:
ST03_514_B71_6.BitInToCheck 		(*  ISK auf Übergabeposition 4*)
END_TRANSITION

TRANSITION Pos4Empty:
NOT ST03_514_B71_6.BitInToCheck  	(*  ISK auf Übergabeposition 4*)
END_TRANSITION

TRANSITION Pos3 Ready:
ST03_514_B71_5.BitInToCheck 	 (* ISK auf Übergabeposition 3 *)
END_TRANSITION

TRANSITION Pos3Full:
ST03_514_B71_5.BitInToCheck	 	(*  ISK auf Übergabeposition 3*)
END_TRANSITION

TRANSITION State Ok:
ST03_515_Y72_5.State=STATE_OK 	(* Übergabeposition Stopper 2 AST/GST *)
END_TRANSITION

TRANSITION Pos4Empty:
NOT ST03_514_B71_6.BitInToCheck  	(*  ISK auf Übergabeposition 4*)
END_TRANSITION

TRANSITION State Ok:
ST03_515_Y72_6.State=STATE_OK 	(* Übergabeposition Stopper 3 AST/GST *)
END_TRANSITION

TRANSITION Pos4 Ready:
ST03_514_B71_6.BitInToCheck  OR		 (* ISK auf Übergabeposition 4 *)
Delay.Q
END_TRANSITION

TRANSITION Po4Full:
ST03_514_B71_6.BitInToCheck 		(*  ISK auf Übergabeposition 4*)
END_TRANSITION

TRANSITION State Ok:
ST03_515_Y72_6.State=STATE_OK 	(* Übergabeposition Stopper 3 AST/GST *)
END_TRANSITION
END_PROGRAM

(* POU Stations/ST_03_Ruestsaetze/ST_03_SFCs/Zufuehrungen/ST03_7pol_Wendeeinheit, SFC *)
 PROGRAM ST03_7pol_Wendeeinheit
VAR_OUTPUT
	SFCCurrentPOU			: STRING:='ST03_7pol_Wendeeinheit';
	SFCCurrentStep			: STRING:='';
	FB_CurrentStepHistorie	: FB_CurrentStepHistorie;
	SFCTime					: DINT;
	State   				: StateObject	:= STATE_WAIT;
	Result  				: StateResult;
END_VAR
VAR_INPUT
	Start				:BOOL;
END_VAR
VAR
	MsgOK				: BOOL;
	MsgCancel			: BOOL;
	SFCRun				: BOOL;
	SFCTimeStart		: TIME;
	Delay				: TON;
	(* Userdefinded area *)
	WenderDone			: BOOL;
	OverrideHelp			:DINT;
END_VAR
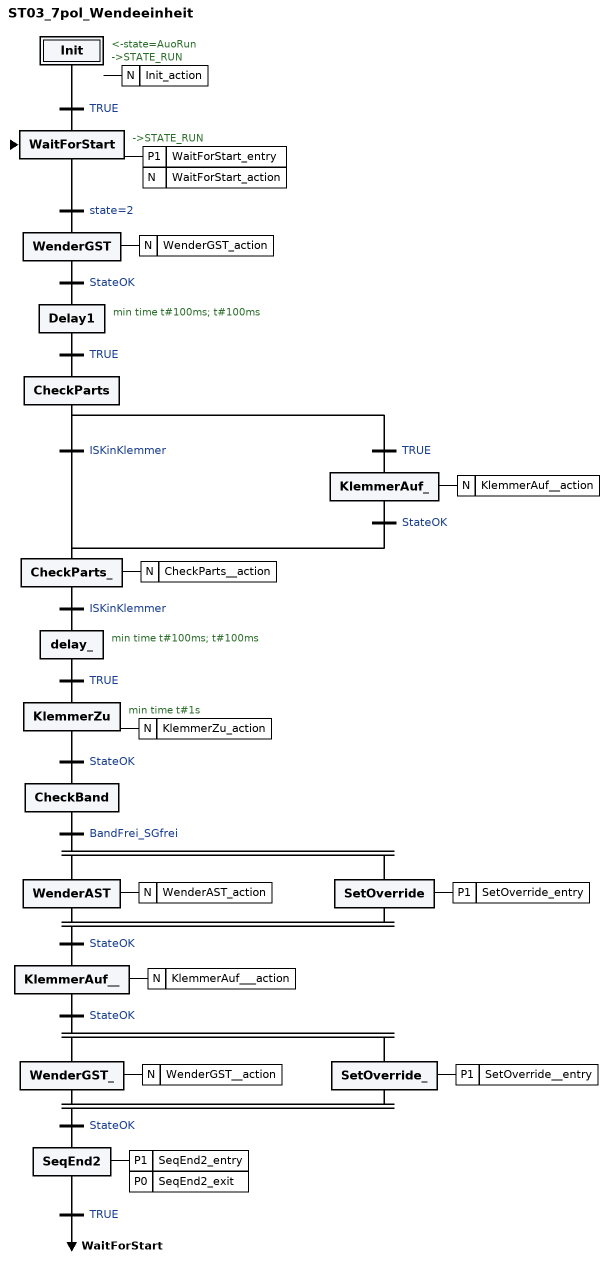
INITIAL_STEP Init: (* <-state=AuoRun / ->STATE_RUN *)
	Init_action(N);
END_STEP
TRANSITION FROM Init TO WaitForStart := TRUE;
END_TRANSITION
STEP WaitForStart: (* ->STATE_RUN *)
	WaitForStart_entry(P1);
	WaitForStart_action(N);
END_STEP
TRANSITION FROM WaitForStart TO WenderGST := state=2;
END_TRANSITION
STEP WenderGST:
	WenderGST_action(N);
END_STEP
TRANSITION FROM WenderGST TO Delay1 := StateOK;
END_TRANSITION
STEP Delay1: (* min time t#100ms; t#100ms *)
END_STEP
TRANSITION FROM Delay1 TO CheckParts := TRUE;
END_TRANSITION
STEP CheckParts:
END_STEP
TRANSITION FROM CheckParts TO CheckParts_ := ISKinKlemmer;
END_TRANSITION
TRANSITION FROM CheckParts TO KlemmerAuf_ := TRUE;
END_TRANSITION
STEP KlemmerAuf_:
	KlemmerAuf__action(N);
END_STEP
TRANSITION FROM KlemmerAuf_ TO CheckParts_ := StateOK;
END_TRANSITION
STEP CheckParts_:
	CheckParts__action(N);
END_STEP
TRANSITION FROM CheckParts_ TO delay_ := ISKinKlemmer;
END_TRANSITION
STEP delay_: (* min time t#100ms; t#100ms *)
END_STEP
TRANSITION FROM delay_ TO KlemmerZu := TRUE;
END_TRANSITION
STEP KlemmerZu: (* min time t#1s *)
	KlemmerZu_action(N);
END_STEP
TRANSITION FROM KlemmerZu TO CheckBand := StateOK;
END_TRANSITION
STEP CheckBand:
END_STEP
TRANSITION FROM CheckBand TO (WenderAST, SetOverride) := BandFrei_SGfrei;
END_TRANSITION
STEP WenderAST:
	WenderAST_action(N);
END_STEP
STEP SetOverride:
	SetOverride_entry(P1);
END_STEP
TRANSITION FROM (WenderAST, SetOverride) TO KlemmerAuf__ := StateOK;
END_TRANSITION
STEP KlemmerAuf__:
	KlemmerAuf___action(N);
END_STEP
TRANSITION FROM KlemmerAuf__ TO (WenderGST_, SetOverride_) := StateOK;
END_TRANSITION
STEP WenderGST_:
	WenderGST__action(N);
END_STEP
STEP SetOverride_:
	SetOverride__entry(P1);
END_STEP
TRANSITION FROM (WenderGST_, SetOverride_) TO SeqEnd2 := StateOK;
END_TRANSITION
STEP SeqEnd2:
	SeqEnd2_entry(P1);
	SeqEnd2_exit(P0);
END_STEP
TRANSITION FROM SeqEnd2 TO WaitForStart := TRUE;
END_TRANSITION

ACTION Init_action:
Start:=FALSE;
State:=STATE_WAIT;
MsgOK:=FALSE;
MsgCancel:=FALSE;
SFCRun:=FALSE;
Result:=RESULT_NON;
IF 	OverrideHelp <> 0 THEN
	MP.ST02.Override_Band:=OverrideHelp;
END_IF
END_ACTION

ACTION WaitForStart_entry:
;
END_ACTION

ACTION WaitForStart_action:
IF 	Start   THEN
	State:=STATE_RUN;
	Result:=RESULT_NON;
	SFCTimeStart:=TIME();
	Start:=FALSE;
	WenderDone:=FALSE;
ELSE
	State:=STATE_WAIT;
	MsgOK:=FALSE;
	MsgCancel:=FALSE;
	SFCRun:=FALSE;
END_IF
END_ACTION

ACTION WenderGST_action:
ST03_515_Y72_1.MoveInit:=TRUE;		(* Rinne schwenkern AST/GST *)
END_ACTION

ACTION KlemmerAuf__action:
ST03_515_Y72_0.MoveInit:=TRUE;		(* ISK Klemmer AST/GST *)
END_ACTION

ACTION CheckParts__action:
ProcessMessage01:='1IM6';						(*'warte auf Teil in Vereinzelung*)
END_ACTION

ACTION KlemmerZu_action:
ST03_515_Y72_0.MoveWork:=TRUE;		(* ISK Klemmer AST/GST *)
END_ACTION

ACTION WenderAST_action:
ST03_515_Y72_1.MoveWork:=TRUE;		(* Rinne schwenkern AST/GST *)
END_ACTION

ACTION SetOverride_entry:
IF 	MP.ST02.Override_Band > 10 THEN
	OverrideHelp:=MP.ST02.Override_Band;
	MP.ST02.Override_Band:= 0;
END_IF
END_ACTION

ACTION KlemmerAuf___action:
ST03_515_Y72_0.MoveInit:=TRUE;
END_ACTION

ACTION WenderGST__action:
ST03_515_Y72_1.MoveInit:=TRUE;		(* Rinne schwenkern AST/GST *)
END_ACTION

ACTION SetOverride__entry:
MP.ST02.Override_Band:=OverrideHelp;
END_ACTION

ACTION SeqEnd2_entry:
WenderDone:=TRUE;
END_ACTION

ACTION SeqEnd2_exit:
WenderDone:=FALSE;
END_ACTION

TRANSITION StateOK:
ST03_515_Y72_1.State = STATE_OK			 (* Rinne schwenkern AST/GST *)
AND gTipImp
END_TRANSITION

TRANSITION ISKinKlemmer:
ST03_512_XG1.BitInToCheck 	(* ISK in Klemmer *)
AND gTipImp
END_TRANSITION

TRANSITION StateOK:
ST03_515_Y72_0.State = STATE_OK		(*   ISK Klemmer AST/GST *)
AND gTipImp
END_TRANSITION

TRANSITION ISKinKlemmer:
ST03_512_XG1.BitInToCheck AND 	(* ISK in Klemmer *)
gTipImp
END_TRANSITION

TRANSITION StateOK:
ST03_515_Y72_0.State = STATE_OK			(* ISK Klemmer AST/GST *)
AND gTipImp
END_TRANSITION

TRANSITION BandFrei_SGfrei:
ST03_514_B71_7.BitInToCheck  	(* Führungsschiene frei zum schwenken *)
AND (ST00_73_K4.BitInToCheck OR ST02_S1_40K01.BitInToCheck)		(*Schnittstelle Freigabe von Spritzmaschine (nur für Anlagen ohne Rundtisch)*)
AND gTipImp
END_TRANSITION

TRANSITION StateOK:
ST03_515_Y72_1.State = STATE_OK 	(* Förderband  Zuführung Vereinzelner Wender AST/GST *)
AND gTipImp
END_TRANSITION

TRANSITION StateOK:
ST03_515_Y72_0.State = STATE_OK	(* ISK Klemmer AST/GST *)
AND gTipImp
END_TRANSITION

TRANSITION StateOK:
ST03_515_Y72_1.State = STATE_OK 	(* Rinne schwenkern AST/GST *)
AND gTipImp
END_TRANSITION
END_PROGRAM

(* POU Stations/ST_03_Ruestsaetze/ST_03_SFCs/Zufuehrungen/ST03_9pol_Wendeeinheit, SFC *)
 PROGRAM ST03_9pol_Wendeeinheit
VAR_OUTPUT
	SFCCurrentPOU			: STRING:='ST03_7pol_Wendeeinheit';
	SFCCurrentStep			: STRING:='';
	FB_CurrentStepHistorie	: FB_CurrentStepHistorie;
	SFCTime					: DINT;
	State   				: StateObject	:= STATE_WAIT;
	Result  				: StateResult;
END_VAR
VAR_INPUT
	Start				:BOOL;
END_VAR
VAR
	MsgOK				: BOOL;
	MsgCancel			: BOOL;
	SFCRun				: BOOL;
	SFCTimeStart		: TIME;
	Delay				: TON;
	(* Userdefinded area *)
	WenderDone			: BOOL;
	OverrideHelp			:DINT;
END_VAR
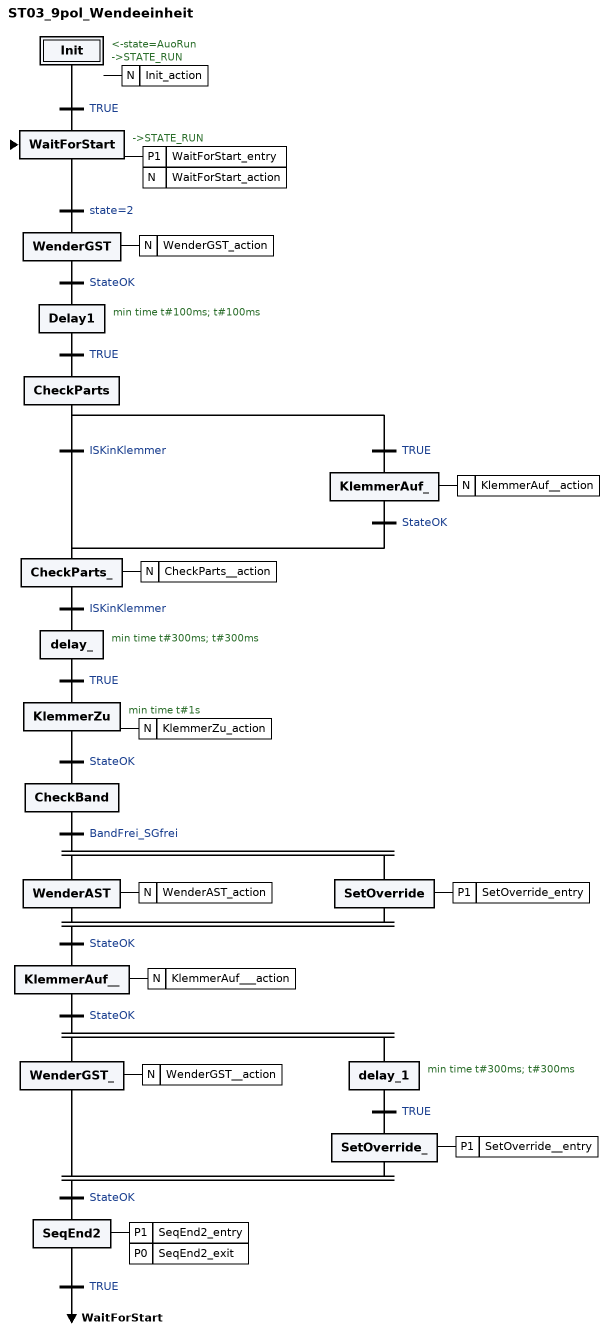
INITIAL_STEP Init: (* <-state=AuoRun / ->STATE_RUN *)
	Init_action(N);
END_STEP
TRANSITION FROM Init TO WaitForStart := TRUE;
END_TRANSITION
STEP WaitForStart: (* ->STATE_RUN *)
	WaitForStart_entry(P1);
	WaitForStart_action(N);
END_STEP
TRANSITION FROM WaitForStart TO WenderGST := state=2;
END_TRANSITION
STEP WenderGST:
	WenderGST_action(N);
END_STEP
TRANSITION FROM WenderGST TO Delay1 := StateOK;
END_TRANSITION
STEP Delay1: (* min time t#100ms; t#100ms *)
END_STEP
TRANSITION FROM Delay1 TO CheckParts := TRUE;
END_TRANSITION
STEP CheckParts:
END_STEP
TRANSITION FROM CheckParts TO CheckParts_ := ISKinKlemmer;
END_TRANSITION
TRANSITION FROM CheckParts TO KlemmerAuf_ := TRUE;
END_TRANSITION
STEP KlemmerAuf_:
	KlemmerAuf__action(N);
END_STEP
TRANSITION FROM KlemmerAuf_ TO CheckParts_ := StateOK;
END_TRANSITION
STEP CheckParts_:
	CheckParts__action(N);
END_STEP
TRANSITION FROM CheckParts_ TO delay_ := ISKinKlemmer;
END_TRANSITION
STEP delay_: (* min time t#300ms; t#300ms *)
END_STEP
TRANSITION FROM delay_ TO KlemmerZu := TRUE;
END_TRANSITION
STEP KlemmerZu: (* min time t#1s *)
	KlemmerZu_action(N);
END_STEP
TRANSITION FROM KlemmerZu TO CheckBand := StateOK;
END_TRANSITION
STEP CheckBand:
END_STEP
TRANSITION FROM CheckBand TO (WenderAST, SetOverride) := BandFrei_SGfrei;
END_TRANSITION
STEP WenderAST:
	WenderAST_action(N);
END_STEP
STEP SetOverride:
	SetOverride_entry(P1);
END_STEP
TRANSITION FROM (WenderAST, SetOverride) TO KlemmerAuf__ := StateOK;
END_TRANSITION
STEP KlemmerAuf__:
	KlemmerAuf___action(N);
END_STEP
TRANSITION FROM KlemmerAuf__ TO (WenderGST_, delay_1) := StateOK;
END_TRANSITION
STEP WenderGST_:
	WenderGST__action(N);
END_STEP
STEP delay_1: (* min time t#300ms; t#300ms *)
END_STEP
TRANSITION FROM delay_1 TO SetOverride_ := TRUE;
END_TRANSITION
STEP SetOverride_:
	SetOverride__entry(P1);
END_STEP
TRANSITION FROM (WenderGST_, SetOverride_) TO SeqEnd2 := StateOK;
END_TRANSITION
STEP SeqEnd2:
	SeqEnd2_entry(P1);
	SeqEnd2_exit(P0);
END_STEP
TRANSITION FROM SeqEnd2 TO WaitForStart := TRUE;
END_TRANSITION

ACTION Init_action:
Start:=FALSE;
State:=STATE_WAIT;
MsgOK:=FALSE;
MsgCancel:=FALSE;
SFCRun:=FALSE;
Result:=RESULT_NON;
IF 	OverrideHelp <> 0 THEN
	MP.ST02.Override_Band:=OverrideHelp;
END_IF
END_ACTION

ACTION WaitForStart_entry:
;
END_ACTION

ACTION WaitForStart_action:
IF 	Start   THEN
	State:=STATE_RUN;
	Result:=RESULT_NON;
	SFCTimeStart:=TIME();
	Start:=FALSE;
	WenderDone:=FALSE;
ELSE
	State:=STATE_WAIT;
	MsgOK:=FALSE;
	MsgCancel:=FALSE;
	SFCRun:=FALSE;
END_IF
END_ACTION

ACTION WenderGST_action:
ST03_515_Y72_1.MoveInit:=TRUE;		(* Rinne schwenkern AST/GST *)
END_ACTION

ACTION KlemmerAuf__action:
ST03_515_Y72_0.MoveInit:=TRUE;		(* ISK Klemmer AST/GST *)
END_ACTION

ACTION CheckParts__action:
ProcessMessage01:='1IM6';						(*'warte auf Teil in Vereinzelung*)
END_ACTION

ACTION KlemmerZu_action:
ST03_515_Y72_0.MoveWork:=TRUE;		(* ISK Klemmer AST/GST *)
END_ACTION

ACTION WenderAST_action:
ST03_515_Y72_1.MoveWork:=TRUE;		(* Rinne schwenkern AST/GST *)
END_ACTION

ACTION SetOverride_entry:
IF 	MP.ST02.Override_Band > 10 THEN
	OverrideHelp:=MP.ST02.Override_Band;
	MP.ST02.Override_Band:= 0;
END_IF
END_ACTION

ACTION KlemmerAuf___action:
ST03_515_Y72_0.MoveInit:=TRUE;
END_ACTION

ACTION WenderGST__action:
ST03_515_Y72_1.MoveInit:=TRUE;		(* Rinne schwenkern AST/GST *)
END_ACTION

ACTION SetOverride__entry:
MP.ST02.Override_Band:=OverrideHelp;
END_ACTION

ACTION SeqEnd2_entry:
WenderDone:=TRUE;
END_ACTION

ACTION SeqEnd2_exit:
WenderDone:=FALSE;
END_ACTION

TRANSITION StateOK:
ST03_515_Y72_1.State = STATE_OK			 (* Rinne schwenkern AST/GST *)
AND gTipImp
END_TRANSITION

TRANSITION ISKinKlemmer:
ST03_512_XG1.BitInToCheck 	(* ISK in Klemmer *)
AND gTipImp
END_TRANSITION

TRANSITION StateOK:
ST03_515_Y72_0.State = STATE_OK		(*   ISK Klemmer AST/GST *)
AND gTipImp
END_TRANSITION

TRANSITION ISKinKlemmer:
ST03_512_XG1.BitInToCheck AND 	(* ISK in Klemmer *)
gTipImp
END_TRANSITION

TRANSITION StateOK:
ST03_515_Y72_0.State = STATE_OK			(* ISK Klemmer AST/GST *)
AND gTipImp
END_TRANSITION

TRANSITION BandFrei_SGfrei:
ST03_514_B71_7.BitInToCheck  	(* Führungsschiene frei zum schwenken *)
AND (ST00_73_K4.BitInToCheck OR ST02_S1_40K01.BitInToCheck)		(*Schnittstelle Freigabe von Spritzmaschine (nur für Anlagen ohne Rundtisch)*)
AND gTipImp
END_TRANSITION

TRANSITION StateOK:
ST03_515_Y72_1.State = STATE_OK 	(* Förderband  Zuführung Vereinzelner Wender AST/GST *)
AND gTipImp
END_TRANSITION

TRANSITION StateOK:
ST03_515_Y72_0.State = STATE_OK	(* ISK Klemmer AST/GST *)
AND gTipImp
END_TRANSITION

TRANSITION StateOK:
ST03_515_Y72_1.State = STATE_OK 	(* Rinne schwenkern AST/GST *)
AND gTipImp
END_TRANSITION
END_PROGRAM

(* POU Stations/ST_03_Ruestsaetze/ST_03_SFCs/Zufuehrungen/ST03_88polAMG_Zufuehrung, SFC *)
 PROGRAM ST03_88polAMG_Zufuehrung
VAR_OUTPUT
	SFCCurrentPOU		: STRING:='ST03_88polAMG_Zufuehrung';
	SFCCurrentStep		: STRING:='';
	FB_CurrentStepHistorie: FB_CurrentStepHistorie;
	SFCTime				: DINT;
	State   			: StateObject	:= STATE_WAIT;
	Result  			: StateResult;
END_VAR
VAR_INPUT
	Start				:BOOL;
END_VAR
VAR
	MsgOK				: BOOL;
	MsgCancel			: BOOL;
	SFCRun				: BOOL;
	SFCTimeStart		: TIME;
	Delay				: TON;
	(* Userdefinded area *)

END_VAR
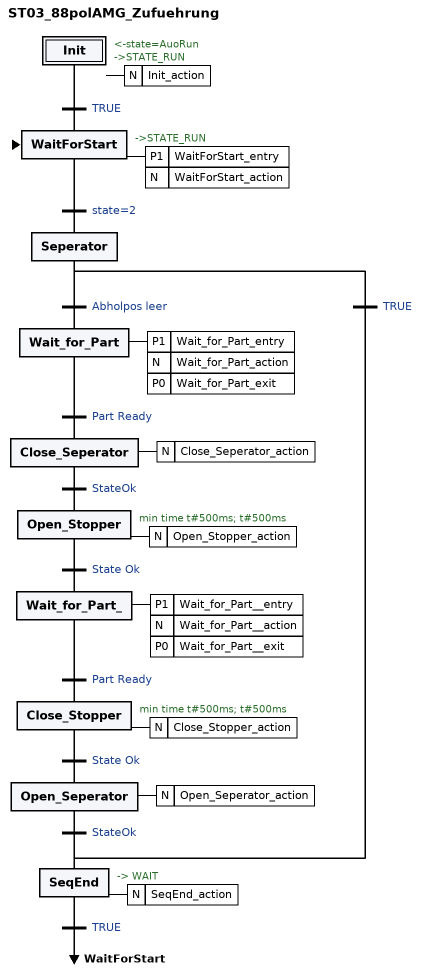
INITIAL_STEP Init: (* <-state=AuoRun / ->STATE_RUN *)
	Init_action(N);
END_STEP
TRANSITION FROM Init TO WaitForStart := TRUE;
END_TRANSITION
STEP WaitForStart: (* ->STATE_RUN *)
	WaitForStart_entry(P1);
	WaitForStart_action(N);
END_STEP
TRANSITION FROM WaitForStart TO Seperator := state=2;
END_TRANSITION
STEP Seperator:
END_STEP
TRANSITION FROM Seperator TO Wait_for_Part := Abholpos leer;
END_TRANSITION
TRANSITION FROM Seperator TO SeqEnd := TRUE;
END_TRANSITION
STEP Wait_for_Part:
	Wait_for_Part_entry(P1);
	Wait_for_Part_action(N);
	Wait_for_Part_exit(P0);
END_STEP
TRANSITION FROM Wait_for_Part TO Close_Seperator := Part Ready;
END_TRANSITION
STEP Close_Seperator:
	Close_Seperator_action(N);
END_STEP
TRANSITION FROM Close_Seperator TO Open_Stopper := StateOk;
END_TRANSITION
STEP Open_Stopper: (* min time t#500ms; t#500ms *)
	Open_Stopper_action(N);
END_STEP
TRANSITION FROM Open_Stopper TO Wait_for_Part_ := State Ok;
END_TRANSITION
STEP Wait_for_Part_:
	Wait_for_Part__entry(P1);
	Wait_for_Part__action(N);
	Wait_for_Part__exit(P0);
END_STEP
TRANSITION FROM Wait_for_Part_ TO Close_Stopper := Part Ready;
END_TRANSITION
STEP Close_Stopper: (* min time t#500ms; t#500ms *)
	Close_Stopper_action(N);
END_STEP
TRANSITION FROM Close_Stopper TO Open_Seperator := State Ok;
END_TRANSITION
STEP Open_Seperator:
	Open_Seperator_action(N);
END_STEP
TRANSITION FROM Open_Seperator TO SeqEnd := StateOk;
END_TRANSITION
STEP SeqEnd: (* -> WAIT *)
	SeqEnd_action(N);
END_STEP
TRANSITION FROM SeqEnd TO WaitForStart := TRUE;
END_TRANSITION

ACTION Init_action:
Start:=FALSE;
State:=STATE_WAIT;
MsgOK:=FALSE;
MsgCancel:=FALSE;
SFCRun:=FALSE;
Result:=RESULT_NON;
END_ACTION

ACTION WaitForStart_entry:
;
END_ACTION

ACTION WaitForStart_action:
IF 	Start   THEN
	State:=STATE_RUN;
	Result:=RESULT_NON;
	SFCTimeStart:=TIME();
	Start:=FALSE;
ELSE
	State:=STATE_WAIT;
	MsgOK:=FALSE;
	MsgCancel:=FALSE;
	SFCRun:=FALSE;
END_IF
END_ACTION

ACTION Wait_for_Part_entry:
ProcessMessage01:='';
Delay.IN:=FALSE;
Delay();
END_ACTION

ACTION Wait_for_Part_action:
ProcessMessage01:='1IM9';(*warte auf Teil in Stopper*)
Delay.IN:=ST03_521_B69_6.BitInToCheck; 		(*  ISK an stopper.*)
Delay.PT:=T#500ms;
Delay();
END_ACTION

ACTION Wait_for_Part_exit:
ProcessMessage01:='';
END_ACTION

ACTION Close_Seperator_action:
ST03_522_Y70_1.MoveWork:=TRUE;		(* Zuführung Vereinzler AST/GST *)
END_ACTION

ACTION Open_Stopper_action:
ST03_522_Y70_2.MoveWork:=TRUE;		(* Züführung Stopper AST/GST *)
END_ACTION

ACTION Wait_for_Part__entry:
ProcessMessage01:='';
Delay.IN:=FALSE;
Delay();
END_ACTION

ACTION Wait_for_Part__action:
ProcessMessage01:='1IM10';(*warte auf Teil in Abholposition*)
Delay.IN:=	ST03_Init_AbholPos.RoboPos31 OR
			ST03_Init_AbholPos.RoboPos35;
Delay.PT:=T#500ms;
Delay();
END_ACTION

ACTION Wait_for_Part__exit:
ProcessMessage01:='';
END_ACTION

ACTION Close_Stopper_action:
ST03_522_Y70_2.MoveInit:=TRUE;		(* Züführung Stopper AST/GST *)
END_ACTION

ACTION Open_Seperator_action:
ST03_522_Y70_1.MoveInit:=TRUE;		(* Zuführung Vereinzler AST/GST *)
END_ACTION

ACTION SeqEnd_action:
SFCTime:=TIME_TO_DINT(TIME()-SFCTimeStart);
State:=STATE_WAIT;
END_ACTION

TRANSITION Abholpos leer:
NOT  ST03_521_B69_7.BitInToCheck AND		(*  ISK Lageerkennung links*)
NOT  ST03_522_B70_0.BitInToCheck 		(*  ISK Lageerkennung rechts*)
END_TRANSITION

TRANSITION Part Ready:
Delay.Q AND
NOT ST03_521_B69_7.BitInToCheck	AND		(*  ISK Lageerkennung links*)
NOT ST03_522_B70_0.BitInToCheck	AND		(*  ISK Lageerkennung rechts*)
ST03_521_B69_6.BitInToCheck	AND				(*  ISK anwesend am Stoper*)
Robot01.ActualArea <> 4
END_TRANSITION

TRANSITION StateOk:
ST03_522_Y70_1.State=STATE_OK 	(* Zuführung Vereinzler AST/GST *)
END_TRANSITION

TRANSITION State Ok:
ST03_522_Y70_2.State=STATE_OK 	(* Züführung Stopper AST/GST *)
END_TRANSITION

TRANSITION Part Ready:
Delay.Q AND
Robot01.ActualArea <> 4
END_TRANSITION

TRANSITION State Ok:
ST03_522_Y70_2.State=STATE_OK 	(*Züführung Stopper AST/GST *)
END_TRANSITION

TRANSITION StateOk:
ST03_522_Y70_1.State=STATE_OK 	(* Zuführung Vereinzler AST/GST *)
END_TRANSITION
END_PROGRAM

(* POU Stations/ST_03_Ruestsaetze/ST_03_SFCs/Zufuehrungen/ST03_120pol_Zufuehrung, SFC *)
 PROGRAM ST03_120pol_Zufuehrung
VAR_OUTPUT
	SFCCurrentPOU		: STRING:='ST03_120pol_Zufuehrung';
	SFCCurrentStep		: STRING:='';
	FB_CurrentStepHistorie: FB_CurrentStepHistorie;
	SFCTime				: DINT;
	State   			: StateObject	:= STATE_WAIT;
	Result  			: StateResult;
END_VAR
VAR_INPUT
	Start				:BOOL;
END_VAR
VAR
	MsgOK				: BOOL;
	MsgCancel			: BOOL;
	SFCRun				: BOOL;
	SFCTimeStart		: TIME;
	Delay				: TON;
	(* Userdefinded area *)

END_VAR
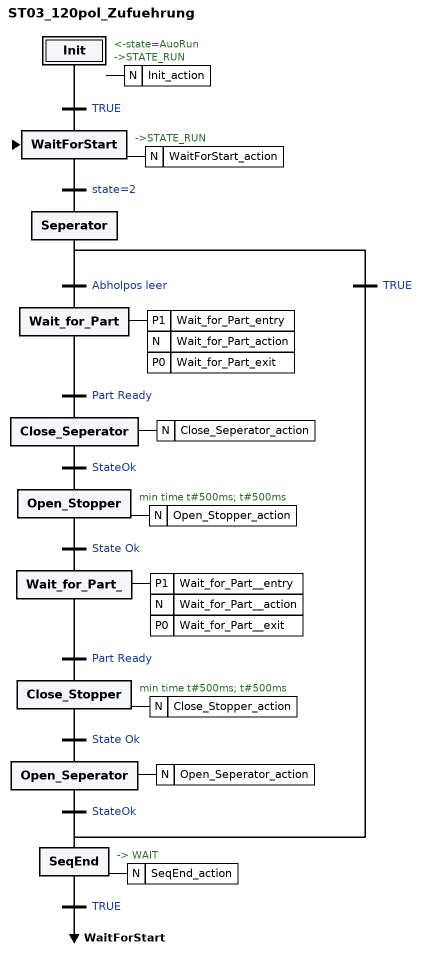
INITIAL_STEP Init: (* <-state=AuoRun / ->STATE_RUN *)
	Init_action(N);
END_STEP
TRANSITION FROM Init TO WaitForStart := TRUE;
END_TRANSITION
STEP WaitForStart: (* ->STATE_RUN *)
	WaitForStart_action(N);
END_STEP
TRANSITION FROM WaitForStart TO Seperator := state=2;
END_TRANSITION
STEP Seperator:
END_STEP
TRANSITION FROM Seperator TO Wait_for_Part := Abholpos leer;
END_TRANSITION
TRANSITION FROM Seperator TO SeqEnd := TRUE;
END_TRANSITION
STEP Wait_for_Part:
	Wait_for_Part_entry(P1);
	Wait_for_Part_action(N);
	Wait_for_Part_exit(P0);
END_STEP
TRANSITION FROM Wait_for_Part TO Close_Seperator := Part Ready;
END_TRANSITION
STEP Close_Seperator:
	Close_Seperator_action(N);
END_STEP
TRANSITION FROM Close_Seperator TO Open_Stopper := StateOk;
END_TRANSITION
STEP Open_Stopper: (* min time t#500ms; t#500ms *)
	Open_Stopper_action(N);
END_STEP
TRANSITION FROM Open_Stopper TO Wait_for_Part_ := State Ok;
END_TRANSITION
STEP Wait_for_Part_:
	Wait_for_Part__entry(P1);
	Wait_for_Part__action(N);
	Wait_for_Part__exit(P0);
END_STEP
TRANSITION FROM Wait_for_Part_ TO Close_Stopper := Part Ready;
END_TRANSITION
STEP Close_Stopper: (* min time t#500ms; t#500ms *)
	Close_Stopper_action(N);
END_STEP
TRANSITION FROM Close_Stopper TO Open_Seperator := State Ok;
END_TRANSITION
STEP Open_Seperator:
	Open_Seperator_action(N);
END_STEP
TRANSITION FROM Open_Seperator TO SeqEnd := StateOk;
END_TRANSITION
STEP SeqEnd: (* -> WAIT *)
	SeqEnd_action(N);
END_STEP
TRANSITION FROM SeqEnd TO WaitForStart := TRUE;
END_TRANSITION

ACTION Init_action:
Start:=FALSE;
State:=STATE_WAIT;
MsgOK:=FALSE;
MsgCancel:=FALSE;
SFCRun:=FALSE;
Result:=RESULT_NON;
END_ACTION

ACTION WaitForStart_action:
IF 	Start   THEN
	State:=STATE_RUN;
	Result:=RESULT_NON;
	SFCTimeStart:=TIME();
	Start:=FALSE;
ELSE
	State:=STATE_WAIT;
	MsgOK:=FALSE;
	MsgCancel:=FALSE;
	SFCRun:=FALSE;
END_IF
END_ACTION

ACTION Wait_for_Part_entry:
ProcessMessage01:='';
Delay.IN:=FALSE;
Delay();
END_ACTION

ACTION Wait_for_Part_action:
ProcessMessage01:='1IM9';(*warte auf Teil in Stopper*)
Delay.IN:=ST03_531_B69_6.BitInToCheck; 		(*  ISK an stopper.*)
Delay.PT:=T#500ms;
Delay();
END_ACTION

ACTION Wait_for_Part_exit:
ProcessMessage01:='';
END_ACTION

ACTION Close_Seperator_action:
ST03_532_Y70_1.MoveWork:=TRUE;		(*Zuführung Vereinzler AST/GST *)
END_ACTION

ACTION Open_Stopper_action:
ST03_532_Y70_2.MoveWork:=TRUE;		(* Züführung Stopper AST/GST *)
END_ACTION

ACTION Wait_for_Part__entry:
ProcessMessage01:='';
Delay.IN:=FALSE;
Delay();
END_ACTION

ACTION Wait_for_Part__action:
ProcessMessage01:='1IM10';(*warte auf Teil in Abholposition*)
Delay.IN:=	ST03_Init_AbholPos.RoboPos31 OR
			ST03_Init_AbholPos.RoboPos35;
Delay.PT:=T#500ms;
Delay();
END_ACTION

ACTION Wait_for_Part__exit:
ProcessMessage01:='';
END_ACTION

ACTION Close_Stopper_action:
ST03_532_Y70_2.MoveInit:=TRUE;		(* Züführung Stopper AST/GST *)
END_ACTION

ACTION Open_Seperator_action:
ST03_532_Y70_1.MoveInit:=TRUE;		(* Zuführung Vereinzler AST/GST *)
END_ACTION

ACTION SeqEnd_action:
SFCTime:=TIME_TO_DINT(TIME()-SFCTimeStart);
State:=STATE_WAIT;
END_ACTION

TRANSITION Abholpos leer:
NOT  ST03_531_B69_7.BitInToCheck AND	(*ISK rechts Lageerkennung*)
NOT ST03_532_B70_0.BitInToCheck		(*ISK links Lageerkennung*)
END_TRANSITION

TRANSITION Part Ready:
Delay.Q AND
NOT ST03_531_B69_7.BitInToCheck	AND		(*ISK rechts Lageerkennung*)
NOT ST03_532_B70_0.BitInToCheck	AND		(*ISK links Lageerkennung*)
ST03_531_B69_6.BitInToCheck	AND			(*ISK anwesend am Stoper*)
Robot01.ActualArea <> 4
END_TRANSITION

TRANSITION StateOk:
ST03_532_Y70_1.State=STATE_OK 	(* Zuführung Vereinzler AST/GST *)
END_TRANSITION

TRANSITION State Ok:
ST03_532_Y70_2.State=STATE_OK 	(* Züführung Stopper AST/GST *)
END_TRANSITION

TRANSITION Part Ready:
Delay.Q AND
Robot01.ActualArea <> 4
END_TRANSITION

TRANSITION State Ok:
ST03_532_Y70_2.State=STATE_OK 	(*Züführung Stopper AST/GST *)
END_TRANSITION

TRANSITION StateOk:
ST03_532_Y70_1.State=STATE_OK 	(* Zuführung Vereinzler AST/GST *)
END_TRANSITION
END_PROGRAM

(* POU Stations/ST_03_Ruestsaetze/ST_03_SFCs/Zufuehrungen/ST03_21pol_Zufuehrung, SFC *)
 PROGRAM ST03_21pol_Zufuehrung
VAR_OUTPUT
	SFCCurrentPOU		: STRING:='ST03_21pol_Zufuehrung';
	SFCCurrentStep		: STRING:='';
	FB_CurrentStepHistorie: FB_CurrentStepHistorie;
	SFCTime				: DINT;
	State   			: StateObject	:= STATE_WAIT;
	Result  			: StateResult;
END_VAR
VAR_INPUT
	Start				:BOOL;
END_VAR
VAR
	MsgOK				: BOOL;
	MsgCancel			: BOOL;
	SFCRun				: BOOL;
	SFCTimeStart		: TIME;
	Delay				: TON;
	(* Userdefinded area *)

END_VAR
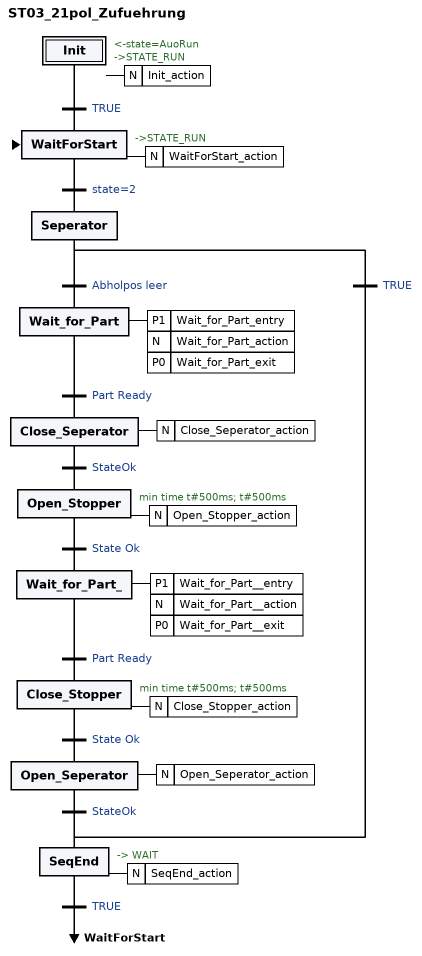
INITIAL_STEP Init: (* <-state=AuoRun / ->STATE_RUN *)
	Init_action(N);
END_STEP
TRANSITION FROM Init TO WaitForStart := TRUE;
END_TRANSITION
STEP WaitForStart: (* ->STATE_RUN *)
	WaitForStart_action(N);
END_STEP
TRANSITION FROM WaitForStart TO Seperator := state=2;
END_TRANSITION
STEP Seperator:
END_STEP
TRANSITION FROM Seperator TO Wait_for_Part := Abholpos leer;
END_TRANSITION
TRANSITION FROM Seperator TO SeqEnd := TRUE;
END_TRANSITION
STEP Wait_for_Part:
	Wait_for_Part_entry(P1);
	Wait_for_Part_action(N);
	Wait_for_Part_exit(P0);
END_STEP
TRANSITION FROM Wait_for_Part TO Close_Seperator := Part Ready;
END_TRANSITION
STEP Close_Seperator:
	Close_Seperator_action(N);
END_STEP
TRANSITION FROM Close_Seperator TO Open_Stopper := StateOk;
END_TRANSITION
STEP Open_Stopper: (* min time t#500ms; t#500ms *)
	Open_Stopper_action(N);
END_STEP
TRANSITION FROM Open_Stopper TO Wait_for_Part_ := State Ok;
END_TRANSITION
STEP Wait_for_Part_:
	Wait_for_Part__entry(P1);
	Wait_for_Part__action(N);
	Wait_for_Part__exit(P0);
END_STEP
TRANSITION FROM Wait_for_Part_ TO Close_Stopper := Part Ready;
END_TRANSITION
STEP Close_Stopper: (* min time t#500ms; t#500ms *)
	Close_Stopper_action(N);
END_STEP
TRANSITION FROM Close_Stopper TO Open_Seperator := State Ok;
END_TRANSITION
STEP Open_Seperator:
	Open_Seperator_action(N);
END_STEP
TRANSITION FROM Open_Seperator TO SeqEnd := StateOk;
END_TRANSITION
STEP SeqEnd: (* -> WAIT *)
	SeqEnd_action(N);
END_STEP
TRANSITION FROM SeqEnd TO WaitForStart := TRUE;
END_TRANSITION

ACTION Init_action:
Start:=FALSE;
State:=STATE_WAIT;
MsgOK:=FALSE;
MsgCancel:=FALSE;
SFCRun:=FALSE;
Result:=RESULT_NON;
END_ACTION

ACTION WaitForStart_action:
IF 	Start   THEN
	State:=STATE_RUN;
	Result:=RESULT_NON;
	SFCTimeStart:=TIME();
	Start:=FALSE;
ELSE
	State:=STATE_WAIT;
	MsgOK:=FALSE;
	MsgCancel:=FALSE;
	SFCRun:=FALSE;
END_IF
END_ACTION

ACTION Wait_for_Part_entry:
ProcessMessage01:='';
Delay.IN:=FALSE;
Delay();
END_ACTION

ACTION Wait_for_Part_action:
ProcessMessage01:='1IM9';(*warte auf Teil in Stopper*)
Delay.IN:=ST03_536_B69_6.BitInToCheck; 		(*  ISK an stopper.*)
Delay.PT:=T#500ms;
Delay();
END_ACTION

ACTION Wait_for_Part_exit:
ProcessMessage01:='';
END_ACTION

ACTION Close_Seperator_action:
ST03_537_Y70_1.MoveWork:=TRUE;		(*Zuführung Vereinzler AST/GST *)
END_ACTION

ACTION Open_Stopper_action:
ST03_537_Y70_2.MoveWork:=TRUE;		(* Züführung Stopper AST/GST *)
END_ACTION

ACTION Wait_for_Part__entry:
ProcessMessage01:='';
Delay.IN:=FALSE;
Delay();
END_ACTION

ACTION Wait_for_Part__action:
ProcessMessage01:='1IM10';(*warte auf Teil in Abholposition*)
Delay.IN:=	ST03_Init_AbholPos.RoboPos31 OR
			ST03_Init_AbholPos.RoboPos35;
Delay.PT:=T#500ms;
Delay();
END_ACTION

ACTION Wait_for_Part__exit:
ProcessMessage01:='';
END_ACTION

ACTION Close_Stopper_action:
ST03_537_Y70_2.MoveInit:=TRUE;		(* Züführung Stopper AST/GST *)
END_ACTION

ACTION Open_Seperator_action:
ST03_537_Y70_1.MoveInit:=TRUE;		(* Zuführung Vereinzler AST/GST *)
END_ACTION

ACTION SeqEnd_action:
SFCTime:=TIME_TO_DINT(TIME()-SFCTimeStart);
State:=STATE_WAIT;
END_ACTION

TRANSITION Abholpos leer:
NOT  ST03_536_B69_7.BitInToCheck		(*  ISK anwesend an Abholposition*)
END_TRANSITION

TRANSITION Part Ready:
Delay.Q AND
NOT ST03_536_B69_7.BitInToCheck	AND		(*ISK anwesend an Abholposition*)
NOT ST03_537_B70_0.BitInToCheck	AND		(*ISK Lageerkennung*)
ST03_536_B69_6.BitInToCheck	AND			(*ISK anwesend am Stoper*)
Robot01.ActualArea <> 4
END_TRANSITION

TRANSITION StateOk:
ST03_537_Y70_1.State=STATE_OK 	(* Zuführung Vereinzler AST/GST *)
END_TRANSITION

TRANSITION State Ok:
ST03_537_Y70_2.State=STATE_OK 	(* Züführung Stopper AST/GST *)
END_TRANSITION

TRANSITION Part Ready:
Delay.Q AND
Robot01.ActualArea <> 4
END_TRANSITION

TRANSITION State Ok:
ST03_537_Y70_2.State=STATE_OK 	(*Züführung Stopper AST/GST *)
END_TRANSITION

TRANSITION StateOk:
ST03_537_Y70_1.State=STATE_OK 	(* Zuführung Vereinzler AST/GST *)
END_TRANSITION
END_PROGRAM

(* POU Stations/ST_03_Ruestsaetze/ST_03_SFCs/Zufuehrungen/ST03_191pol_Zufuehrung, SFC *)
 PROGRAM ST03_191pol_Zufuehrung
VAR_OUTPUT
	SFCCurrentPOU		: STRING:='ST03_191pol_Zufuehrung';
	SFCCurrentStep		: STRING:='';
	FB_CurrentStepHistorie: FB_CurrentStepHistorie;
	SFCTime				: DINT;
	State   			: StateObject	:= STATE_WAIT;
	Result  			: StateResult;
END_VAR
VAR_INPUT
	Start				:BOOL;
END_VAR
VAR
	MsgOK				: BOOL;
	MsgCancel			: BOOL;
	SFCRun				: BOOL;
	SFCTimeStart		: TIME;
	Delay				: TON;
	(* Userdefinded area *)

END_VAR
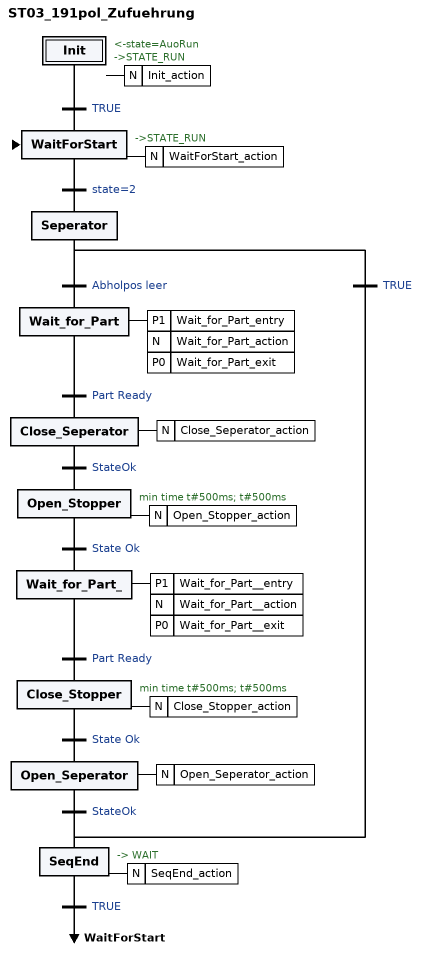
INITIAL_STEP Init: (* <-state=AuoRun / ->STATE_RUN *)
	Init_action(N);
END_STEP
TRANSITION FROM Init TO WaitForStart := TRUE;
END_TRANSITION
STEP WaitForStart: (* ->STATE_RUN *)
	WaitForStart_action(N);
END_STEP
TRANSITION FROM WaitForStart TO Seperator := state=2;
END_TRANSITION
STEP Seperator:
END_STEP
TRANSITION FROM Seperator TO Wait_for_Part := Abholpos leer;
END_TRANSITION
TRANSITION FROM Seperator TO SeqEnd := TRUE;
END_TRANSITION
STEP Wait_for_Part:
	Wait_for_Part_entry(P1);
	Wait_for_Part_action(N);
	Wait_for_Part_exit(P0);
END_STEP
TRANSITION FROM Wait_for_Part TO Close_Seperator := Part Ready;
END_TRANSITION
STEP Close_Seperator:
	Close_Seperator_action(N);
END_STEP
TRANSITION FROM Close_Seperator TO Open_Stopper := StateOk;
END_TRANSITION
STEP Open_Stopper: (* min time t#500ms; t#500ms *)
	Open_Stopper_action(N);
END_STEP
TRANSITION FROM Open_Stopper TO Wait_for_Part_ := State Ok;
END_TRANSITION
STEP Wait_for_Part_:
	Wait_for_Part__entry(P1);
	Wait_for_Part__action(N);
	Wait_for_Part__exit(P0);
END_STEP
TRANSITION FROM Wait_for_Part_ TO Close_Stopper := Part Ready;
END_TRANSITION
STEP Close_Stopper: (* min time t#500ms; t#500ms *)
	Close_Stopper_action(N);
END_STEP
TRANSITION FROM Close_Stopper TO Open_Seperator := State Ok;
END_TRANSITION
STEP Open_Seperator:
	Open_Seperator_action(N);
END_STEP
TRANSITION FROM Open_Seperator TO SeqEnd := StateOk;
END_TRANSITION
STEP SeqEnd: (* -> WAIT *)
	SeqEnd_action(N);
END_STEP
TRANSITION FROM SeqEnd TO WaitForStart := TRUE;
END_TRANSITION

ACTION Init_action:
Start:=FALSE;
State:=STATE_WAIT;
MsgOK:=FALSE;
MsgCancel:=FALSE;
SFCRun:=FALSE;
Result:=RESULT_NON;
END_ACTION

ACTION WaitForStart_action:
IF 	Start   THEN
	State:=STATE_RUN;
	Result:=RESULT_NON;
	SFCTimeStart:=TIME();
	Start:=FALSE;
ELSE
	State:=STATE_WAIT;
	MsgOK:=FALSE;
	MsgCancel:=FALSE;
	SFCRun:=FALSE;
END_IF
END_ACTION

ACTION Wait_for_Part_entry:
ProcessMessage01:='';
Delay.IN:=FALSE;
Delay();
END_ACTION

ACTION Wait_for_Part_action:
ProcessMessage01:='1IM9';(*warte auf Teil in Stopper*)
Delay.IN:=ST03_541_B69_6.BitInToCheck; 		(*  ISK an stopper.*)
Delay.PT:=T#500ms;
Delay();
END_ACTION

ACTION Wait_for_Part_exit:
ProcessMessage01:='';
END_ACTION

ACTION Close_Seperator_action:
ST03_542_Y70_1.MoveWork:=TRUE;		(*Zuführung Vereinzler AST/GST *)
END_ACTION

ACTION Open_Stopper_action:
ST03_542_Y70_2.MoveWork:=TRUE;		(* Züführung Stopper AST/GST *)
END_ACTION

ACTION Wait_for_Part__entry:
ProcessMessage01:='';
Delay.IN:=FALSE;
Delay();
END_ACTION

ACTION Wait_for_Part__action:
ProcessMessage01:='1IM10';(*warte auf Teil in Abholposition*)
Delay.IN:=	ST03_Init_AbholPos.RoboPos31 OR
			ST03_Init_AbholPos.RoboPos35;
Delay.PT:=T#500ms;
Delay();
END_ACTION

ACTION Wait_for_Part__exit:
ProcessMessage01:='';
END_ACTION

ACTION Close_Stopper_action:
ST03_542_Y70_2.MoveInit:=TRUE;		(* Züführung Stopper AST/GST *)
END_ACTION

ACTION Open_Seperator_action:
ST03_542_Y70_1.MoveInit:=TRUE;		(* Zuführung Vereinzler AST/GST *)
END_ACTION

ACTION SeqEnd_action:
SFCTime:=TIME_TO_DINT(TIME()-SFCTimeStart);
State:=STATE_WAIT;
END_ACTION

TRANSITION Abholpos leer:
NOT ST03_Init_AbholPos.RoboPos31 AND
NOT ST03_Init_AbholPos.RoboPos35
END_TRANSITION

TRANSITION Part Ready:
Delay.Q AND
NOT ST03_541_B69_7.BitInToCheck	AND		(*ISK links Lageerkennung*)
NOT ST03_542_B70_0.BitInToCheck	AND		(*ISK rechts Lageerkennung*)
ST03_541_B69_6.BitInToCheck	AND			(*ISK anwesend am Stoper*)
Robot01.ActualArea <> 4
END_TRANSITION

TRANSITION StateOk:
ST03_542_Y70_1.State=STATE_OK 	(* Zuführung Vereinzler AST/GST *)
END_TRANSITION

TRANSITION State Ok:
ST03_542_Y70_2.State=STATE_OK 	(* Züführung Stopper AST/GST *)
END_TRANSITION

TRANSITION Part Ready:
Delay.Q AND
Robot01.ActualArea <> 4
END_TRANSITION

TRANSITION State Ok:
ST03_542_Y70_2.State=STATE_OK 	(*Züführung Stopper AST/GST *)
END_TRANSITION

TRANSITION StateOk:
ST03_542_Y70_1.State=STATE_OK 	(* Zuführung Vereinzler AST/GST *)
END_TRANSITION
END_PROGRAM

(* POU Stations/ST_03_Ruestsaetze/ST_03_SFCs/Zufuehrungen/ST03_72pol_Zufuehrung, SFC *)
 PROGRAM ST03_72pol_Zufuehrung
VAR_OUTPUT
	SFCCurrentPOU		: STRING:='ST03_72pol_Zufuehrung';
	SFCCurrentStep		: STRING:='';
	FB_CurrentStepHistorie: FB_CurrentStepHistorie;
	SFCTime				: DINT;
	State   			: StateObject	:= STATE_WAIT;
	Result  			: StateResult;
END_VAR
VAR_INPUT
	Start				:BOOL;
END_VAR
VAR
	MsgOK				: BOOL;
	MsgCancel			: BOOL;
	SFCRun				: BOOL;
	SFCTimeStart		: TIME;
	Delay				: TON;
	(* Userdefinded area *)

END_VAR
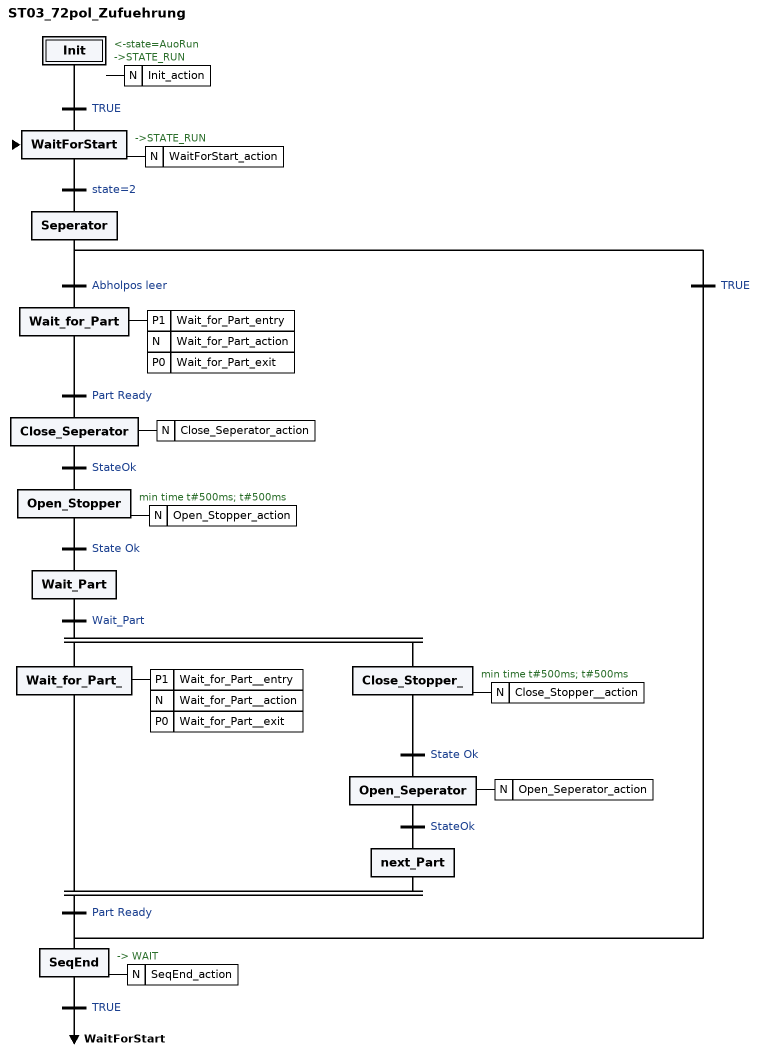
INITIAL_STEP Init: (* <-state=AuoRun / ->STATE_RUN *)
	Init_action(N);
END_STEP
TRANSITION FROM Init TO WaitForStart := TRUE;
END_TRANSITION
STEP WaitForStart: (* ->STATE_RUN *)
	WaitForStart_action(N);
END_STEP
TRANSITION FROM WaitForStart TO Seperator := state=2;
END_TRANSITION
STEP Seperator:
END_STEP
TRANSITION FROM Seperator TO Wait_for_Part := Abholpos leer;
END_TRANSITION
TRANSITION FROM Seperator TO SeqEnd := TRUE;
END_TRANSITION
STEP Wait_for_Part:
	Wait_for_Part_entry(P1);
	Wait_for_Part_action(N);
	Wait_for_Part_exit(P0);
END_STEP
TRANSITION FROM Wait_for_Part TO Close_Seperator := Part Ready;
END_TRANSITION
STEP Close_Seperator:
	Close_Seperator_action(N);
END_STEP
TRANSITION FROM Close_Seperator TO Open_Stopper := StateOk;
END_TRANSITION
STEP Open_Stopper: (* min time t#500ms; t#500ms *)
	Open_Stopper_action(N);
END_STEP
TRANSITION FROM Open_Stopper TO Wait_Part := State Ok;
END_TRANSITION
STEP Wait_Part:
END_STEP
TRANSITION FROM Wait_Part TO (Wait_for_Part_, Close_Stopper_) := Wait_Part;
END_TRANSITION
STEP Wait_for_Part_:
	Wait_for_Part__entry(P1);
	Wait_for_Part__action(N);
	Wait_for_Part__exit(P0);
END_STEP
STEP Close_Stopper_: (* min time t#500ms; t#500ms *)
	Close_Stopper__action(N);
END_STEP
TRANSITION FROM Close_Stopper_ TO Open_Seperator := State Ok;
END_TRANSITION
STEP Open_Seperator:
	Open_Seperator_action(N);
END_STEP
TRANSITION FROM Open_Seperator TO next_Part := StateOk;
END_TRANSITION
STEP next_Part:
END_STEP
TRANSITION FROM (Wait_for_Part_, next_Part) TO SeqEnd := Part Ready;
END_TRANSITION
STEP SeqEnd: (* -> WAIT *)
	SeqEnd_action(N);
END_STEP
TRANSITION FROM SeqEnd TO WaitForStart := TRUE;
END_TRANSITION

ACTION Init_action:
Start:=FALSE;
State:=STATE_WAIT;
MsgOK:=FALSE;
MsgCancel:=FALSE;
SFCRun:=FALSE;
Result:=RESULT_NON;
END_ACTION

ACTION WaitForStart_action:
IF 	Start   THEN
	State:=STATE_RUN;
	Result:=RESULT_NON;
	SFCTimeStart:=TIME();
	Start:=FALSE;
ELSE
	State:=STATE_WAIT;
	MsgOK:=FALSE;
	MsgCancel:=FALSE;
	SFCRun:=FALSE;
END_IF
END_ACTION

ACTION Wait_for_Part_entry:
ProcessMessage01:='';
Delay(IN:=FALSE);
END_ACTION

ACTION Wait_for_Part_action:
ProcessMessage01:='1IM9';(*warte auf Teil in Stopper*)
Delay(	IN:=ST03_546_B69_6.BitInToCheck,		(*  ISK an stopper.*)
		PT:=T#500ms);
END_ACTION

ACTION Wait_for_Part_exit:
ProcessMessage01:='';
Delay(IN:=FALSE);
END_ACTION

ACTION Close_Seperator_action:
ST03_547_Y70_1.MoveWork:=TRUE;		(*Zuführung Vereinzler AST/GST *)
END_ACTION

ACTION Open_Stopper_action:
ST03_547_Y70_2.MoveWork:=TRUE;		(* Züführung Stopper AST/GST *)
END_ACTION

ACTION Wait_for_Part__entry:
ProcessMessage01:='';
Delay(IN:=FALSE);
END_ACTION

ACTION Wait_for_Part__action:
ProcessMessage01:='1IM10';(*warte auf Teil in Abholposition*)
Delay(	IN:=	NOT ST03_Init_AbholPos.RoboPos31 AND
			NOT ST03_Init_AbholPos.RoboPos35,
		PT:=T#500ms);
END_ACTION

ACTION Wait_for_Part__exit:
ProcessMessage01:='';
Delay(IN:=FALSE);
END_ACTION

ACTION Close_Stopper__action:
ST03_547_Y70_2.MoveInit:=TRUE;		(* Züführung Stopper AST/GST *)
END_ACTION

ACTION Open_Seperator_action:
ST03_547_Y70_1.MoveInit:=TRUE;		(* Zuführung Vereinzler AST/GST *)
END_ACTION

ACTION SeqEnd_action:
SFCTime:=TIME_TO_DINT(TIME()-SFCTimeStart);
State:=STATE_WAIT;
END_ACTION

TRANSITION Abholpos leer:
NOT ST03_Init_AbholPos.RoboPos31 AND
NOT ST03_Init_AbholPos.RoboPos35
END_TRANSITION

TRANSITION Part Ready:
Delay.Q AND
NOT ST03_Init_AbholPos.RoboPos31 AND
NOT ST03_Init_AbholPos.RoboPos35 AND
ST03_546_B69_6.BitInToCheck	AND			(*ISK anwesend am Stoper*)
Robot01.ActualArea <> 4
END_TRANSITION

TRANSITION StateOk:
ST03_547_Y70_1.State=STATE_OK 	(* Zuführung Vereinzler AST/GST *)
END_TRANSITION

TRANSITION State Ok:
ST03_547_Y70_2.State=STATE_OK 	(* Züführung Stopper AST/GST *)
END_TRANSITION

TRANSITION Wait_Part:
ST03_Init_AbholPos.RoboPos31 OR
ST03_Init_AbholPos.RoboPos35
END_TRANSITION

TRANSITION State Ok:
ST03_547_Y70_2.State=STATE_OK 	(*Züführung Stopper AST/GST *)
END_TRANSITION

TRANSITION StateOk:
ST03_547_Y70_1.State=STATE_OK 	(* Zuführung Vereinzler AST/GST *)
END_TRANSITION

TRANSITION Part Ready:
Delay.Q AND
Robot01.ActualArea <> 4
END_TRANSITION
END_PROGRAM

(* POU Stations/ST_03_Ruestsaetze/ST_03_SFCs/Zufuehrungen/ST03_48pol_Zufuehrung, SFC *)
 PROGRAM ST03_48pol_Zufuehrung
VAR_OUTPUT
	SFCCurrentPOU		: STRING:='ST03_48pol_Zufuehrung';
	SFCCurrentStep		: STRING:='';
	FB_CurrentStepHistorie: FB_CurrentStepHistorie;
	SFCTime				: DINT;
	State   			: StateObject	:= STATE_WAIT;
	Result  			: StateResult;
END_VAR
VAR_INPUT
	Start				:BOOL;
END_VAR
VAR
	MsgOK				: BOOL;
	MsgCancel			: BOOL;
	SFCRun				: BOOL;
	SFCTimeStart		: TIME;
	Delay				: TON;
	(* Userdefinded area *)

END_VAR
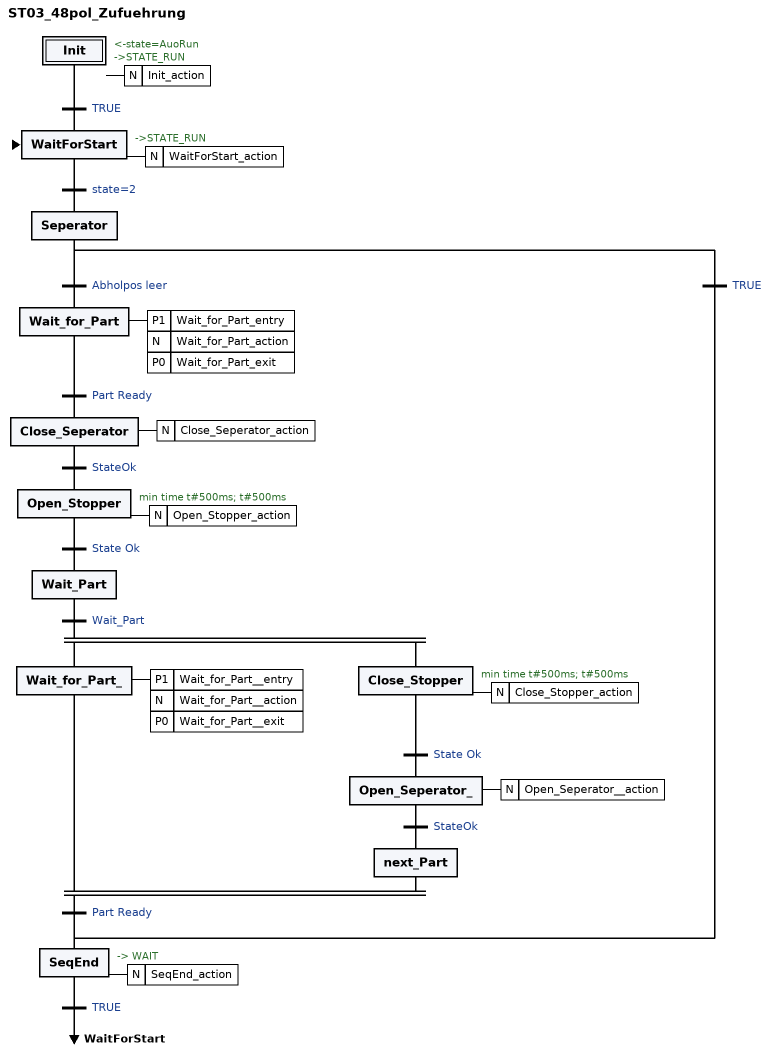
INITIAL_STEP Init: (* <-state=AuoRun / ->STATE_RUN *)
	Init_action(N);
END_STEP
TRANSITION FROM Init TO WaitForStart := TRUE;
END_TRANSITION
STEP WaitForStart: (* ->STATE_RUN *)
	WaitForStart_action(N);
END_STEP
TRANSITION FROM WaitForStart TO Seperator := state=2;
END_TRANSITION
STEP Seperator:
END_STEP
TRANSITION FROM Seperator TO Wait_for_Part := Abholpos leer;
END_TRANSITION
TRANSITION FROM Seperator TO SeqEnd := TRUE;
END_TRANSITION
STEP Wait_for_Part:
	Wait_for_Part_entry(P1);
	Wait_for_Part_action(N);
	Wait_for_Part_exit(P0);
END_STEP
TRANSITION FROM Wait_for_Part TO Close_Seperator := Part Ready;
END_TRANSITION
STEP Close_Seperator:
	Close_Seperator_action(N);
END_STEP
TRANSITION FROM Close_Seperator TO Open_Stopper := StateOk;
END_TRANSITION
STEP Open_Stopper: (* min time t#500ms; t#500ms *)
	Open_Stopper_action(N);
END_STEP
TRANSITION FROM Open_Stopper TO Wait_Part := State Ok;
END_TRANSITION
STEP Wait_Part:
END_STEP
TRANSITION FROM Wait_Part TO (Wait_for_Part_, Close_Stopper) := Wait_Part;
END_TRANSITION
STEP Wait_for_Part_:
	Wait_for_Part__entry(P1);
	Wait_for_Part__action(N);
	Wait_for_Part__exit(P0);
END_STEP
STEP Close_Stopper: (* min time t#500ms; t#500ms *)
	Close_Stopper_action(N);
END_STEP
TRANSITION FROM Close_Stopper TO Open_Seperator_ := State Ok;
END_TRANSITION
STEP Open_Seperator_:
	Open_Seperator__action(N);
END_STEP
TRANSITION FROM Open_Seperator_ TO next_Part := StateOk;
END_TRANSITION
STEP next_Part:
END_STEP
TRANSITION FROM (Wait_for_Part_, next_Part) TO SeqEnd := Part Ready;
END_TRANSITION
STEP SeqEnd: (* -> WAIT *)
	SeqEnd_action(N);
END_STEP
TRANSITION FROM SeqEnd TO WaitForStart := TRUE;
END_TRANSITION

ACTION Init_action:
Start:=FALSE;
State:=STATE_WAIT;
MsgOK:=FALSE;
MsgCancel:=FALSE;
SFCRun:=FALSE;
Result:=RESULT_NON;
END_ACTION

ACTION WaitForStart_action:
IF 	Start   THEN
	State:=STATE_RUN;
	Result:=RESULT_NON;
	SFCTimeStart:=TIME();
	Start:=FALSE;
ELSE
	State:=STATE_WAIT;
	MsgOK:=FALSE;
	MsgCancel:=FALSE;
	SFCRun:=FALSE;
END_IF
END_ACTION

ACTION Wait_for_Part_entry:
ProcessMessage01:='';
Delay(IN:=FALSE);
END_ACTION

ACTION Wait_for_Part_action:
ProcessMessage01:='1IM9';(*warte auf Teil in Stopper*)
Delay(	IN:=ST03_551_B69_6.BitInToCheck, 		(*  ISK an stopper.*)
		PT:=T#500ms);
END_ACTION

ACTION Wait_for_Part_exit:
ProcessMessage01:='';
Delay(IN:=FALSE);
END_ACTION

ACTION Close_Seperator_action:
ST03_552_Y70_1.MoveWork:=TRUE;		(*Zuführung Vereinzler AST/GST *)
END_ACTION

ACTION Open_Stopper_action:
ST03_552_Y70_2.MoveWork:=TRUE;		(* Züführung Stopper AST/GST *)
END_ACTION

ACTION Wait_for_Part__entry:
ProcessMessage01:='';
Delay(IN:=FALSE);
END_ACTION

ACTION Wait_for_Part__action:
ProcessMessage01:='1IM10';(*warte auf Teil in Abholposition*)
Delay(	IN:=	NOT ST03_Init_AbholPos.RoboPos31 AND
			NOT ST03_Init_AbholPos.RoboPos35,
		PT:=T#500ms);
END_ACTION

ACTION Wait_for_Part__exit:
ProcessMessage01:='';
Delay(IN:=FALSE);
END_ACTION

ACTION Close_Stopper_action:
ST03_552_Y70_2.MoveInit:=TRUE;		(* Züführung Stopper AST/GST *)
END_ACTION

ACTION Open_Seperator__action:
ST03_552_Y70_1.MoveInit:=TRUE;		(*Zuführung Vereinzler AST/GST *)
END_ACTION

ACTION SeqEnd_action:
SFCTime:=TIME_TO_DINT(TIME()-SFCTimeStart);
State:=STATE_WAIT;
END_ACTION

TRANSITION Abholpos leer:
NOT ST03_Init_AbholPos.RoboPos31 AND
NOT ST03_Init_AbholPos.RoboPos35
END_TRANSITION

TRANSITION Part Ready:
Delay.Q AND
NOT ST03_Init_AbholPos.RoboPos31 AND
NOT ST03_Init_AbholPos.RoboPos35 AND
ST03_551_B69_6.BitInToCheck	AND			(*ISK anwesend am Stoper*)
Robot01.ActualArea <> 4
END_TRANSITION

TRANSITION StateOk:
ST03_552_Y70_1.State=STATE_OK 	(* Zuführung Vereinzler AST/GST *)
END_TRANSITION

TRANSITION State Ok:
ST03_552_Y70_2.State=STATE_OK 	(* Züführung Stopper AST/GST *)
END_TRANSITION

TRANSITION Wait_Part:
ST03_Init_AbholPos.RoboPos31 OR
ST03_Init_AbholPos.RoboPos35
END_TRANSITION

TRANSITION State Ok:
ST03_552_Y70_2.State=STATE_OK 	(*Züführung Stopper AST/GST *)
END_TRANSITION

TRANSITION StateOk:
ST03_552_Y70_1.State=STATE_OK 	(* Zuführung Vereinzler AST/GST *)
END_TRANSITION

TRANSITION Part Ready:
Delay.Q AND
Robot01.ActualArea <> 4
END_TRANSITION
END_PROGRAM

(* POU Stations/ST_03_Ruestsaetze/ST_03_SFCs/Zufuehrungen/ST03_268pol_Zufuehrung, SFC *)
PROGRAM ST03_268pol_Zufuehrung
VAR_INPUT
	Start					:BOOL;
END_VAR
VAR_OUTPUT
	SFCCurrentPOU			: STRING:='ST03_268pol_Zufuehrung';
	SFCCurrentStep			: STRING:='';
	FB_CurrentStepHistorie: FB_CurrentStepHistorie;
	SFCTime				: DINT;
	State   					: StateObject	:= STATE_WAIT;
	Result  					: ARRAY [1..NO_OF_RESULT] OF StateResult;
	ResultOK				: BOOL;
END_VAR
VAR
	MsgOK				: BOOL;
	MsgCancel			: BOOL;
	SFCRun			: BOOL;
	SFCTimeStart		: TIME;
	Delay				: TON;
	(* Userdefinded area *)

	i					: INT;
	Pos					: INT;
	RepeatCounter		: INT;
	NokCounter			: INT;
	NokCounterPercent	: INT;
  	NokPercent   		: ARRAY[1..100] OF BOOL;
	CamAlwaysOK		:BOOL:=TRUE;		(*schreibt immer OK nur zum Testen*)

END_VAR

VAR CONSTANT
	NO_OF_RESULT	: INT :=2;
END_VAR
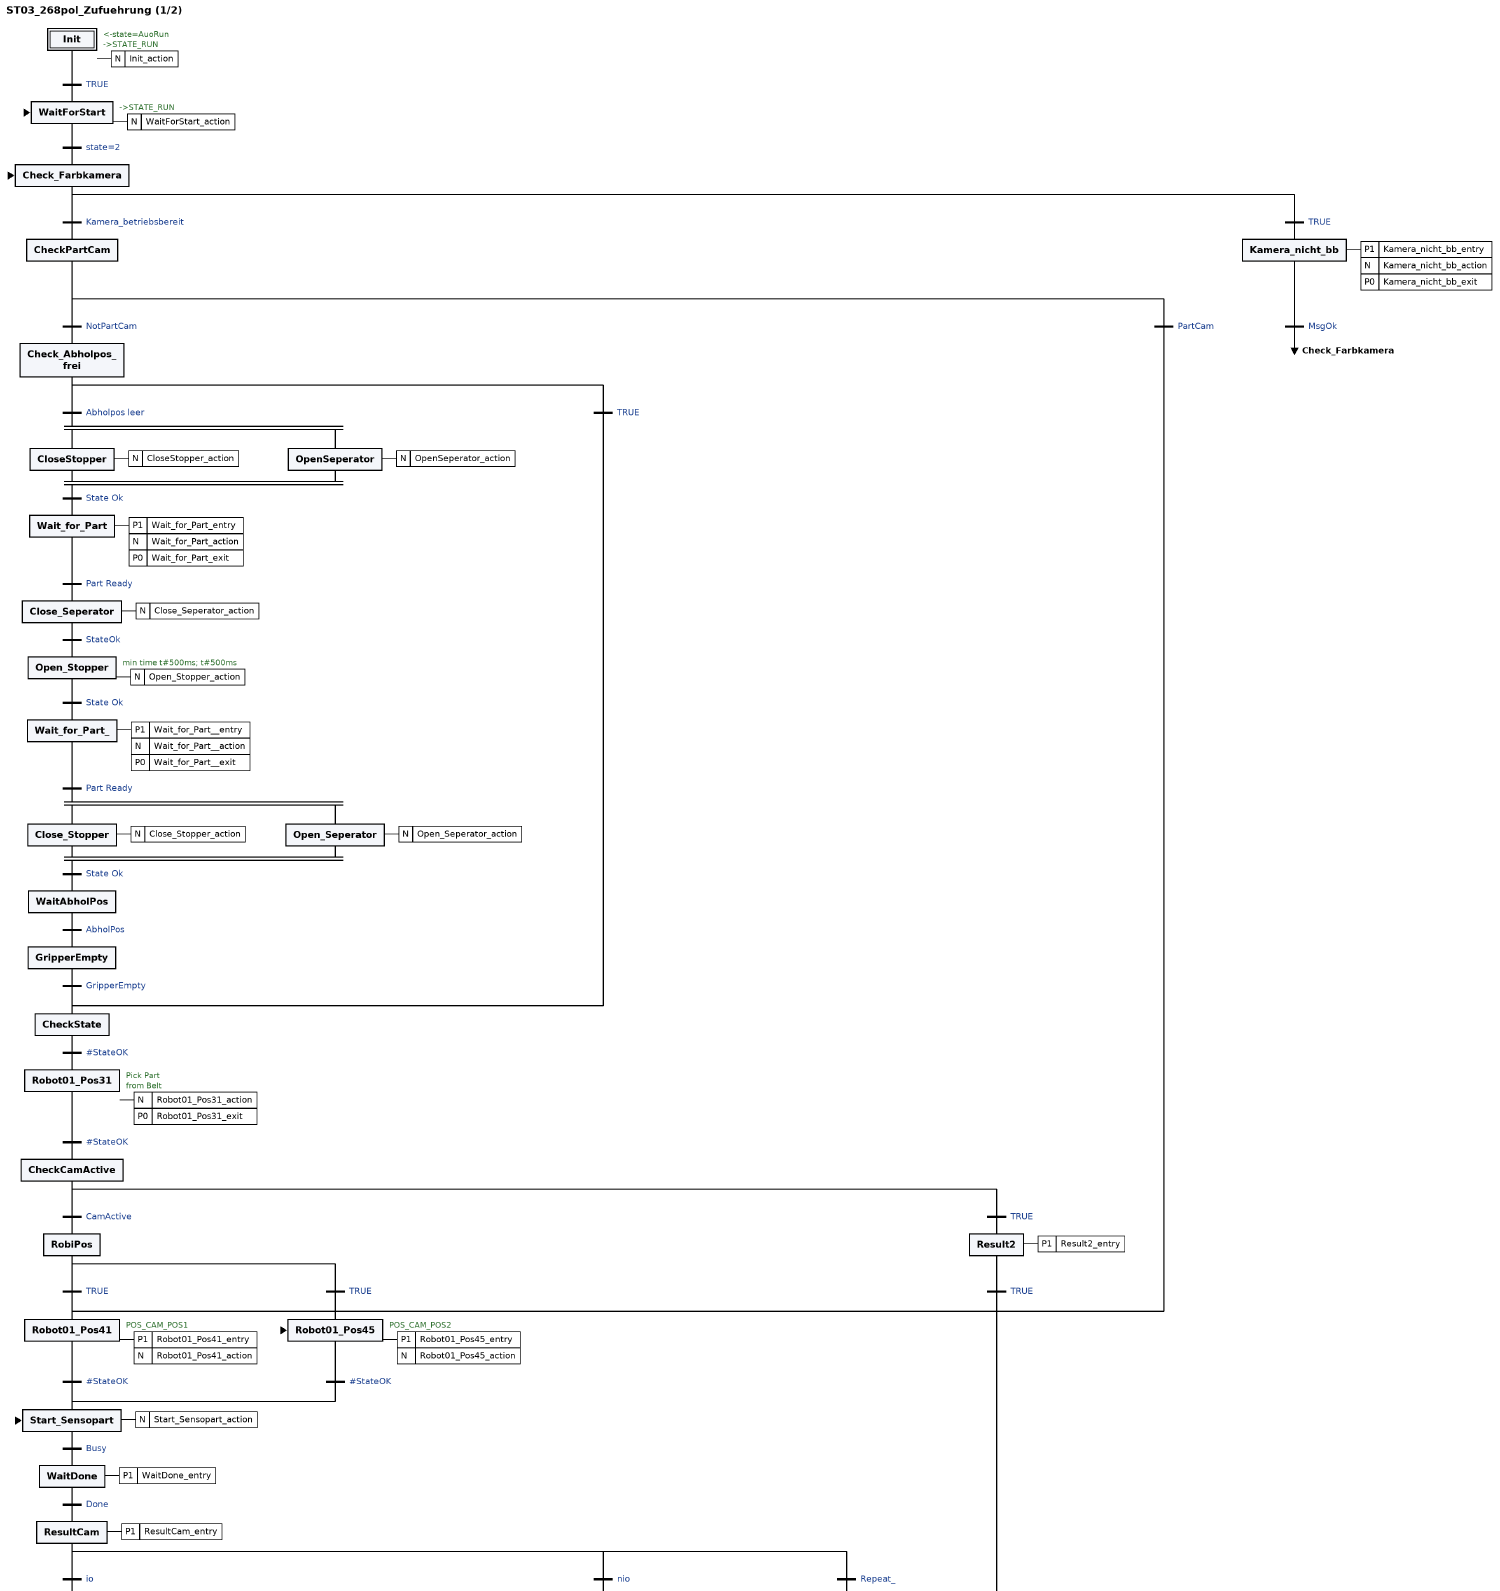
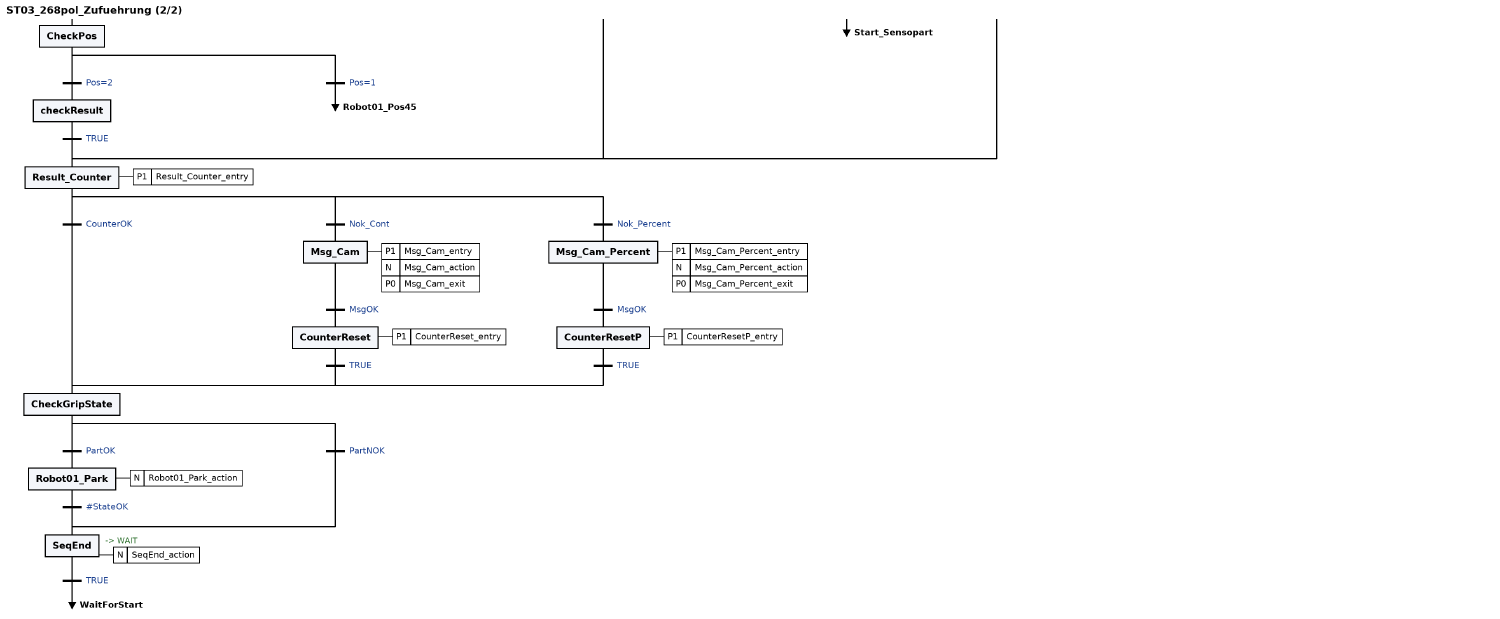
INITIAL_STEP Init: (* <-state=AuoRun / ->STATE_RUN *)
	Init_action(N);
END_STEP
TRANSITION FROM Init TO WaitForStart := TRUE;
END_TRANSITION
STEP WaitForStart: (* ->STATE_RUN *)
	WaitForStart_action(N);
END_STEP
TRANSITION FROM WaitForStart TO Check_Farbkamera := state=2;
END_TRANSITION
STEP Check_Farbkamera:
END_STEP
TRANSITION FROM Check_Farbkamera TO CheckPartCam := Kamera_betriebsbereit;
END_TRANSITION
TRANSITION FROM Check_Farbkamera TO Kamera_nicht_bb := TRUE;
END_TRANSITION
STEP CheckPartCam:
END_STEP
TRANSITION FROM CheckPartCam TO Check_Abholpos_frei := NotPartCam;
END_TRANSITION
TRANSITION FROM CheckPartCam TO Robot01_Pos41 := PartCam;
END_TRANSITION
STEP Check_Abholpos_frei:
END_STEP
TRANSITION FROM Check_Abholpos_frei TO (CloseStopper, OpenSeperator) := Abholpos leer;
END_TRANSITION
TRANSITION FROM Check_Abholpos_frei TO CheckState := TRUE;
END_TRANSITION
STEP CloseStopper:
	CloseStopper_action(N);
END_STEP
STEP OpenSeperator:
	OpenSeperator_action(N);
END_STEP
TRANSITION FROM (CloseStopper, OpenSeperator) TO Wait_for_Part := State Ok;
END_TRANSITION
STEP Kamera_nicht_bb:
	Kamera_nicht_bb_entry(P1);
	Kamera_nicht_bb_action(N);
	Kamera_nicht_bb_exit(P0);
END_STEP
TRANSITION FROM Kamera_nicht_bb TO Check_Farbkamera := MsgOk;
END_TRANSITION
STEP Wait_for_Part:
	Wait_for_Part_entry(P1);
	Wait_for_Part_action(N);
	Wait_for_Part_exit(P0);
END_STEP
TRANSITION FROM Wait_for_Part TO Close_Seperator := Part Ready;
END_TRANSITION
STEP Close_Seperator:
	Close_Seperator_action(N);
END_STEP
TRANSITION FROM Close_Seperator TO Open_Stopper := StateOk;
END_TRANSITION
STEP Open_Stopper: (* min time t#500ms; t#500ms *)
	Open_Stopper_action(N);
END_STEP
TRANSITION FROM Open_Stopper TO Wait_for_Part_ := State Ok;
END_TRANSITION
STEP Wait_for_Part_:
	Wait_for_Part__entry(P1);
	Wait_for_Part__action(N);
	Wait_for_Part__exit(P0);
END_STEP
TRANSITION FROM Wait_for_Part_ TO (Close_Stopper, Open_Seperator) := Part Ready;
END_TRANSITION
STEP Close_Stopper:
	Close_Stopper_action(N);
END_STEP
STEP Open_Seperator:
	Open_Seperator_action(N);
END_STEP
TRANSITION FROM (Close_Stopper, Open_Seperator) TO WaitAbholPos := State Ok;
END_TRANSITION
STEP WaitAbholPos:
END_STEP
TRANSITION FROM WaitAbholPos TO GripperEmpty := AbholPos;
END_TRANSITION
STEP GripperEmpty:
END_STEP
TRANSITION FROM GripperEmpty TO CheckState := GripperEmpty;
END_TRANSITION
STEP CheckState:
END_STEP
TRANSITION FROM CheckState TO Robot01_Pos31 := #StateOK;
END_TRANSITION
STEP Robot01_Pos31: (* Pick Part / from Belt *)
	Robot01_Pos31_action(N);
	Robot01_Pos31_exit(P0);
END_STEP
TRANSITION FROM Robot01_Pos31 TO CheckCamActive := #StateOK;
END_TRANSITION
STEP CheckCamActive:
END_STEP
TRANSITION FROM CheckCamActive TO RobiPos := CamActive;
END_TRANSITION
TRANSITION FROM CheckCamActive TO Result2 := TRUE;
END_TRANSITION
STEP RobiPos:
END_STEP
TRANSITION FROM RobiPos TO Robot01_Pos41 := TRUE;
END_TRANSITION
TRANSITION FROM RobiPos TO Robot01_Pos45 := TRUE;
END_TRANSITION
STEP Robot01_Pos41: (* POS_CAM_POS1 *)
	Robot01_Pos41_entry(P1);
	Robot01_Pos41_action(N);
END_STEP
TRANSITION FROM Robot01_Pos41 TO Start_Sensopart := #StateOK;
END_TRANSITION
STEP Robot01_Pos45: (* POS_CAM_POS2 *)
	Robot01_Pos45_entry(P1);
	Robot01_Pos45_action(N);
END_STEP
TRANSITION FROM Robot01_Pos45 TO Start_Sensopart := #StateOK;
END_TRANSITION
STEP Start_Sensopart:
	Start_Sensopart_action(N);
END_STEP
TRANSITION FROM Start_Sensopart TO WaitDone := Busy;
END_TRANSITION
STEP WaitDone:
	WaitDone_entry(P1);
END_STEP
TRANSITION FROM WaitDone TO ResultCam := Done;
END_TRANSITION
STEP ResultCam:
	ResultCam_entry(P1);
END_STEP
TRANSITION FROM ResultCam TO CheckPos := io;
END_TRANSITION
TRANSITION FROM ResultCam TO Result_Counter := nio;
END_TRANSITION
TRANSITION FROM ResultCam TO Start_Sensopart := Repeat_;
END_TRANSITION
STEP CheckPos:
END_STEP
TRANSITION FROM CheckPos TO checkResult := Pos=2;
END_TRANSITION
TRANSITION FROM CheckPos TO Robot01_Pos45 := Pos=1;
END_TRANSITION
STEP checkResult:
END_STEP
TRANSITION FROM checkResult TO Result_Counter := TRUE;
END_TRANSITION
STEP Result2:
	Result2_entry(P1);
END_STEP
TRANSITION FROM Result2 TO Result_Counter := TRUE;
END_TRANSITION
STEP Result_Counter:
	Result_Counter_entry(P1);
END_STEP
TRANSITION FROM Result_Counter TO CheckGripState := CounterOK;
END_TRANSITION
TRANSITION FROM Result_Counter TO Msg_Cam := Nok_Cont;
END_TRANSITION
TRANSITION FROM Result_Counter TO Msg_Cam_Percent := Nok_Percent;
END_TRANSITION
STEP Msg_Cam:
	Msg_Cam_entry(P1);
	Msg_Cam_action(N);
	Msg_Cam_exit(P0);
END_STEP
TRANSITION FROM Msg_Cam TO CounterReset := MsgOK;
END_TRANSITION
STEP CounterReset:
	CounterReset_entry(P1);
END_STEP
TRANSITION FROM CounterReset TO CheckGripState := TRUE;
END_TRANSITION
STEP Msg_Cam_Percent:
	Msg_Cam_Percent_entry(P1);
	Msg_Cam_Percent_action(N);
	Msg_Cam_Percent_exit(P0);
END_STEP
TRANSITION FROM Msg_Cam_Percent TO CounterResetP := MsgOK;
END_TRANSITION
STEP CounterResetP:
	CounterResetP_entry(P1);
END_STEP
TRANSITION FROM CounterResetP TO CheckGripState := TRUE;
END_TRANSITION
STEP CheckGripState:
END_STEP
TRANSITION FROM CheckGripState TO Robot01_Park := PartOK;
END_TRANSITION
TRANSITION FROM CheckGripState TO SeqEnd := PartNOK;
END_TRANSITION
STEP Robot01_Park:
	Robot01_Park_action(N);
END_STEP
TRANSITION FROM Robot01_Park TO SeqEnd := #StateOK;
END_TRANSITION
STEP SeqEnd: (* -> WAIT *)
	SeqEnd_action(N);
END_STEP
TRANSITION FROM SeqEnd TO WaitForStart := TRUE;
END_TRANSITION

ACTION Init_action:
Start:=FALSE;
State:=STATE_WAIT;
MsgOK:=FALSE;
MsgCancel:=FALSE;
SFCRun:=FALSE;
NokCounter:=0;
i:=1;
Pos:=1;
FOR i:=1 TO NO_OF_RESULT BY 1 DO
	Result[i]:=RESULT_NON;
END_FOR;
END_ACTION

ACTION WaitForStart_action:
i:=1;
IF 	Start   THEN
	State:=STATE_RUN;
	SFCTimeStart:=TIME();
	Start:=FALSE;
	FOR i:=1 TO NO_OF_RESULT BY 1 DO
		Result[i]:=RESULT_NON;
	END_FOR
	Pos:=1;
ELSE
	State:=STATE_WAIT;
	MsgOK:=FALSE;
	MsgCancel:=FALSE;
	SFCRun:=FALSE;
END_IF
END_ACTION

ACTION CloseStopper_action:
ST03_557_Y70_2.MoveInit:=TRUE;		(* Züführung Stopper AST/GST *)
END_ACTION

